END_VAR
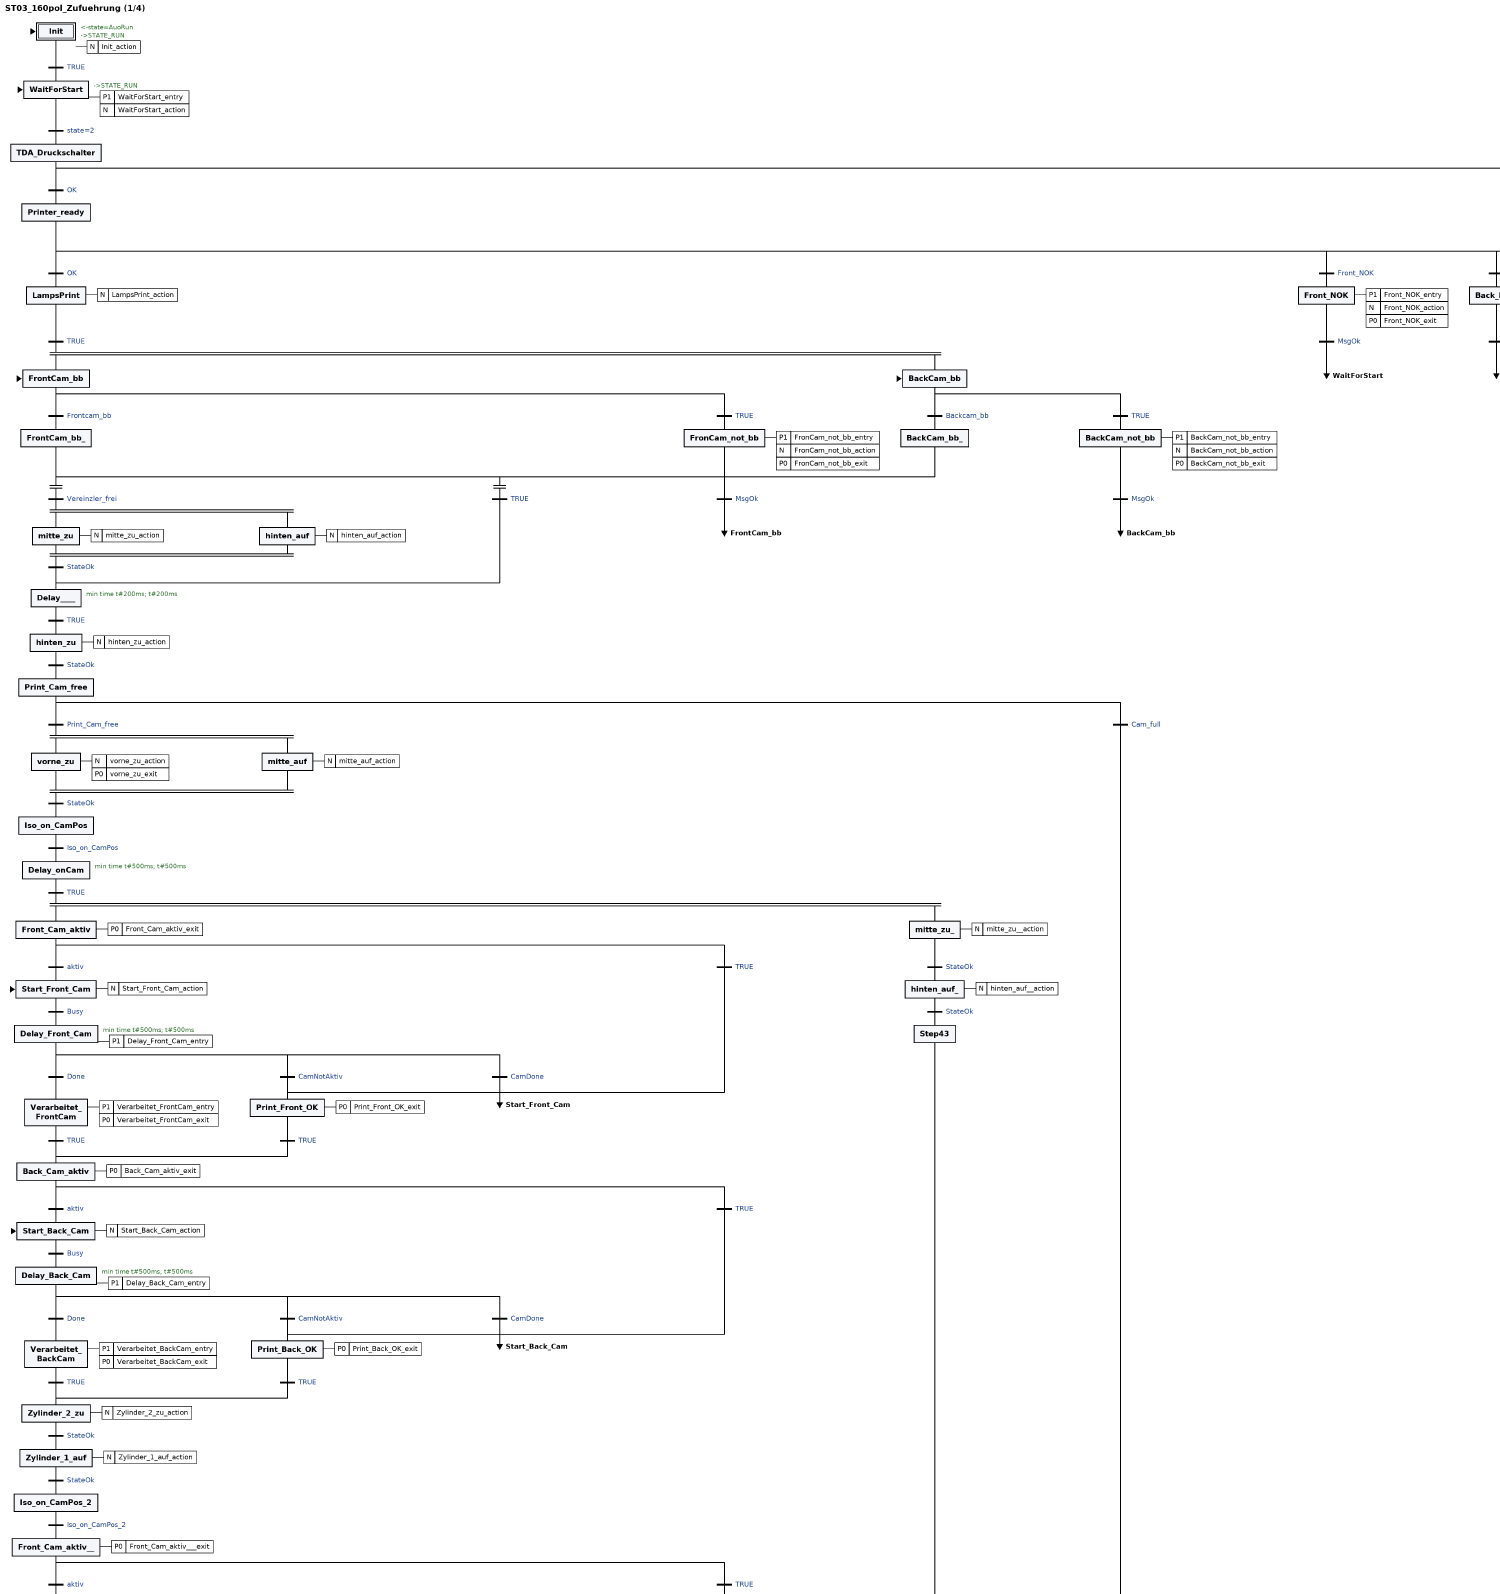
[picture p37: ST03_160pol_Zufuehrung (SFC)]
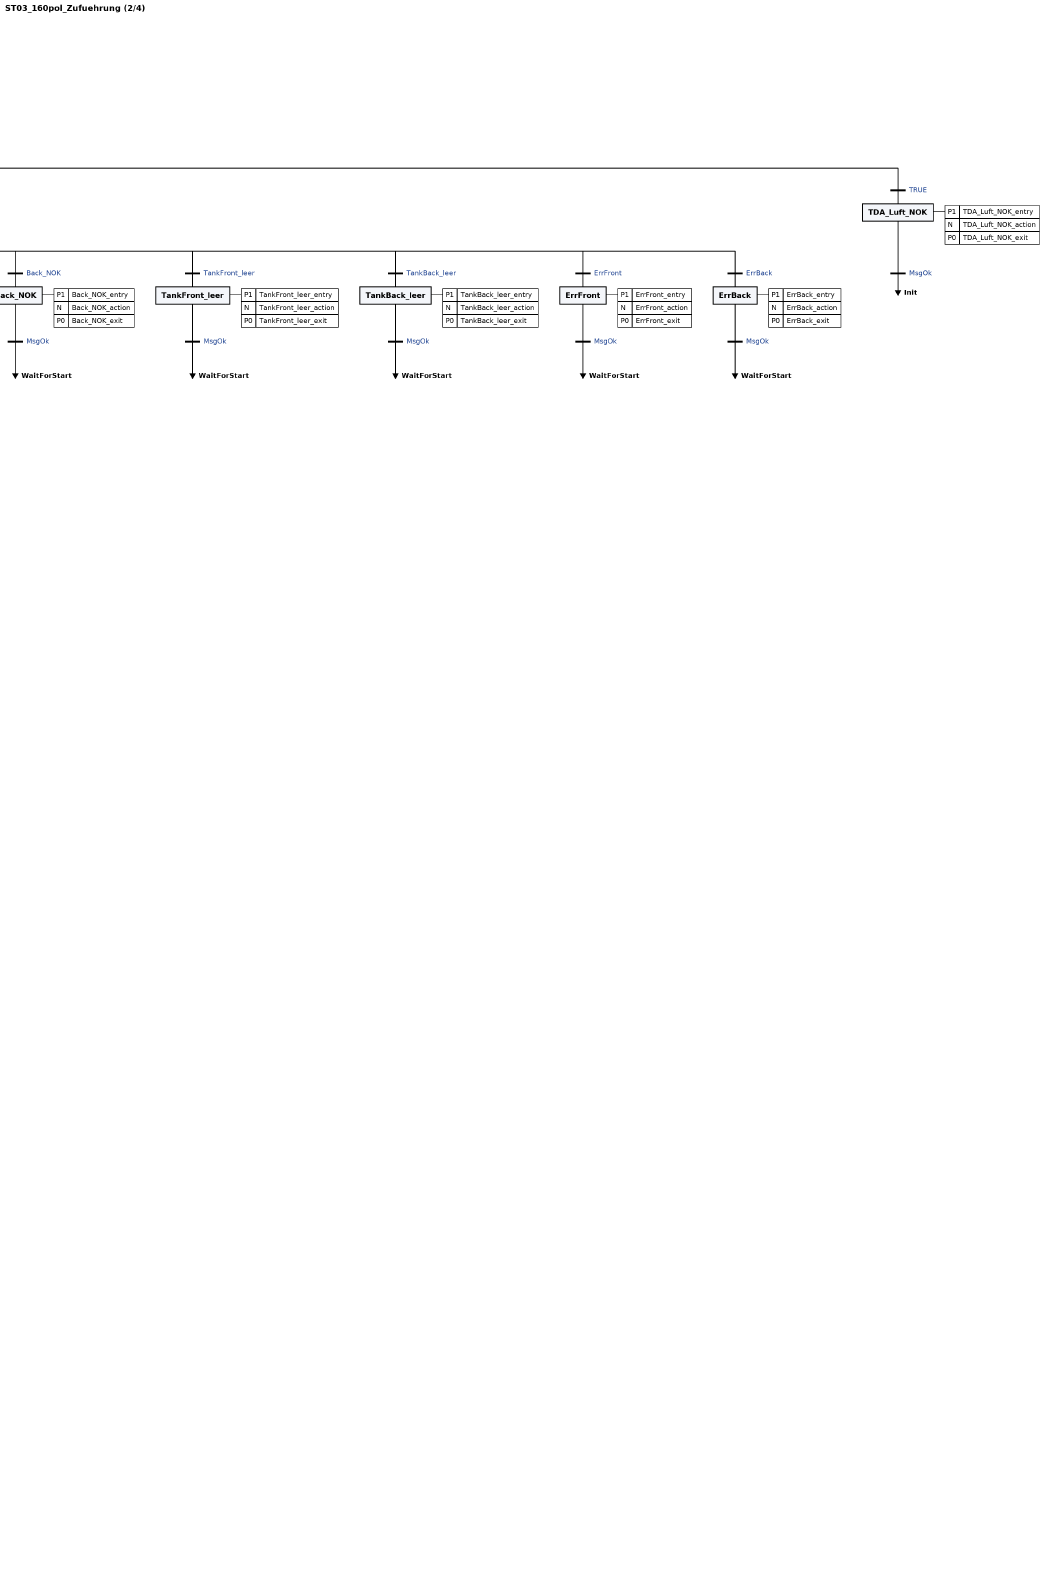
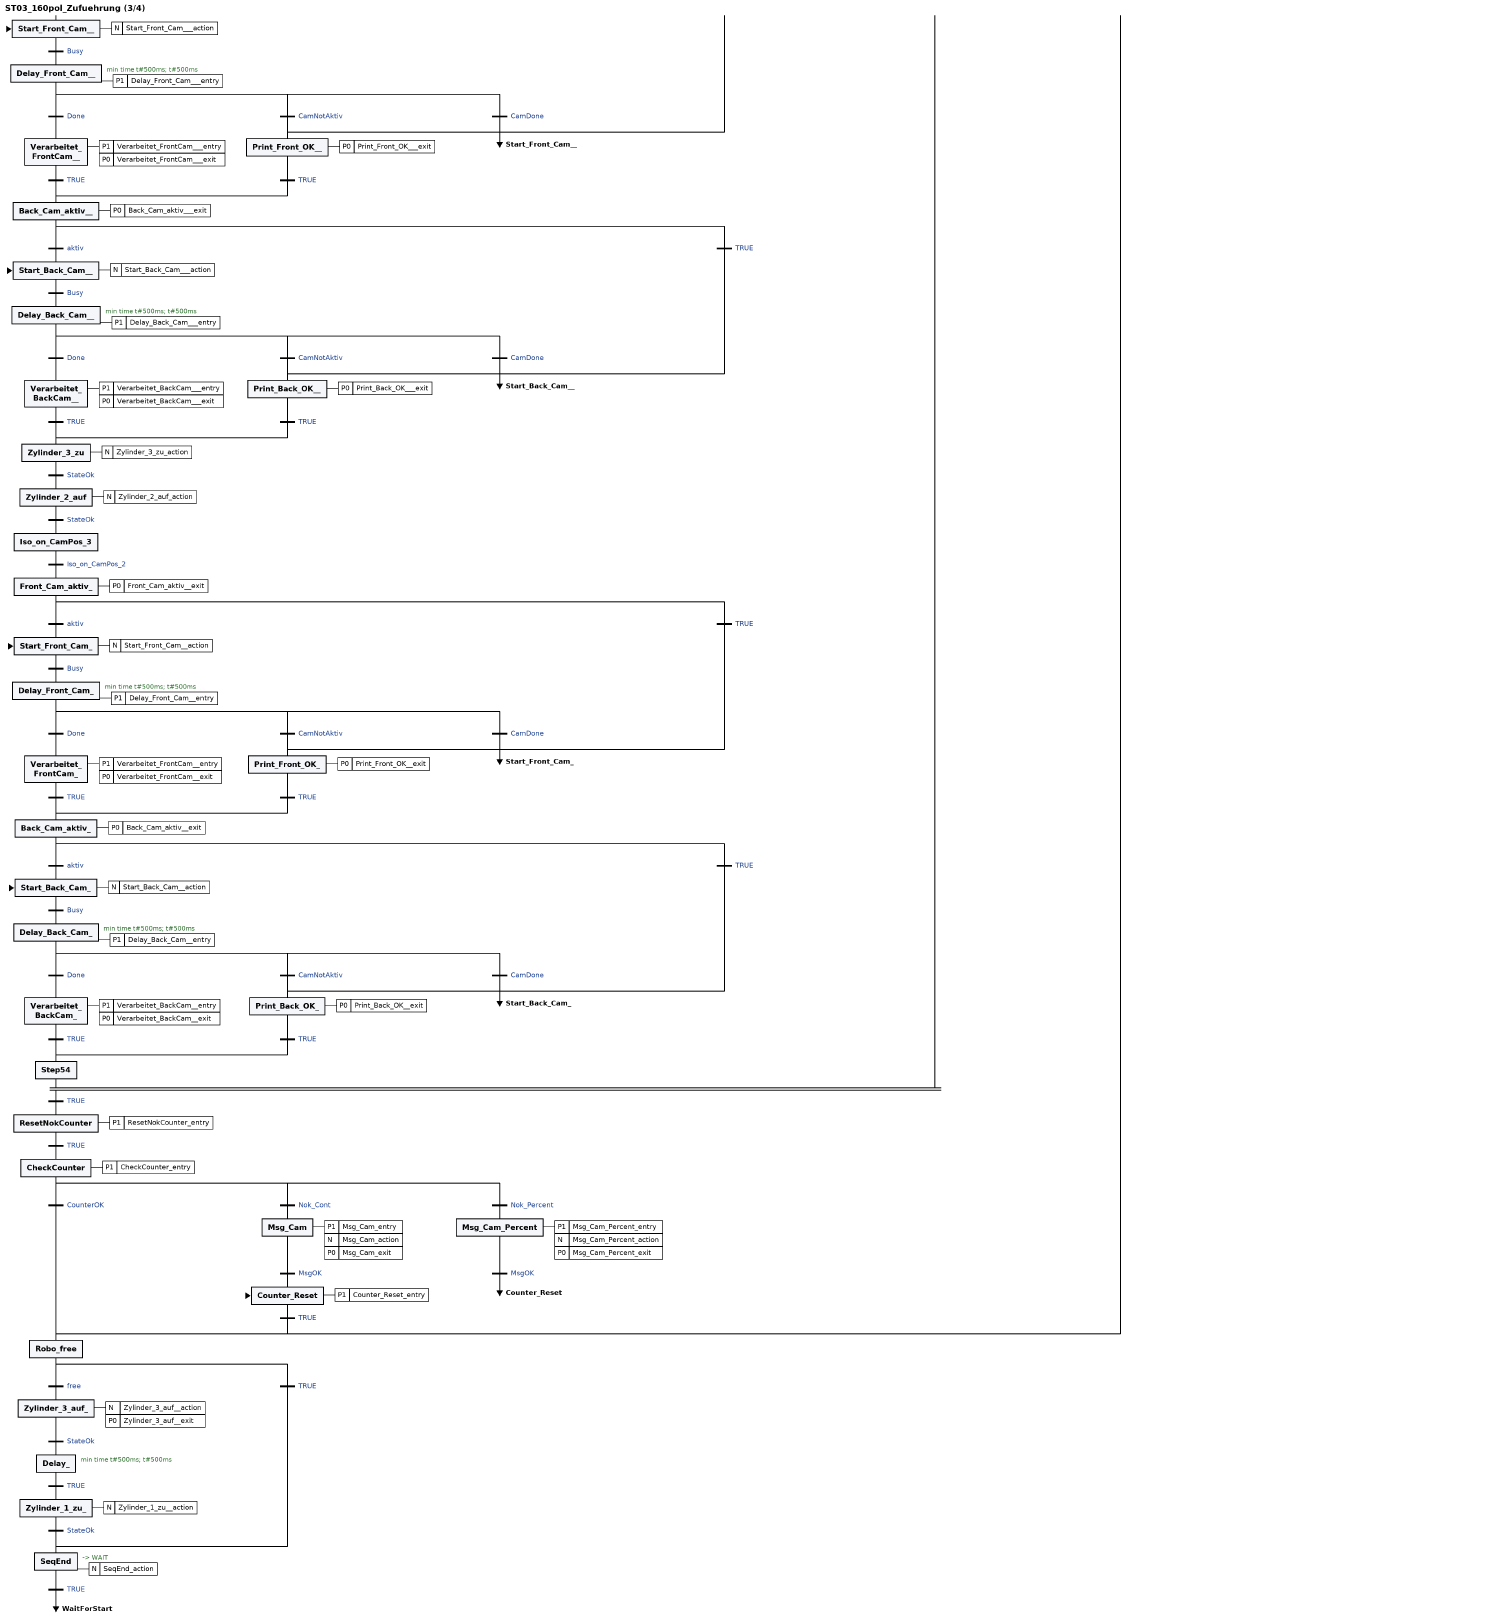
INITIAL_STEP Init: (* <-state=AuoRun / ->STATE_RUN *)
	Init_action(N);
END_STEP
TRANSITION FROM Init TO WaitForStart := TRUE;
END_TRANSITION
STEP WaitForStart: (* ->STATE_RUN *)
	WaitForStart_entry(P1);
	WaitForStart_action(N);
END_STEP
TRANSITION FROM WaitForStart TO TDA_Druckschalter := state=2;
END_TRANSITION
STEP TDA_Druckschalter:
END_STEP
TRANSITION FROM TDA_Druckschalter TO Printer_ready := OK;
END_TRANSITION
TRANSITION FROM TDA_Druckschalter TO TDA_Luft_NOK := TRUE;
END_TRANSITION
STEP TDA_Luft_NOK:
	TDA_Luft_NOK_entry(P1);
	TDA_Luft_NOK_action(N);
	TDA_Luft_NOK_exit(P0);
END_STEP
TRANSITION FROM TDA_Luft_NOK TO Init := MsgOk;
END_TRANSITION
STEP Printer_ready:
END_STEP
TRANSITION FROM Printer_ready TO LampsPrint := OK;
END_TRANSITION
TRANSITION FROM Printer_ready TO Front_NOK := Front_NOK;
END_TRANSITION
TRANSITION FROM Printer_ready TO Back_NOK := Back_NOK;
END_TRANSITION
TRANSITION FROM Printer_ready TO TankFront_leer := TankFront_leer;
END_TRANSITION
TRANSITION FROM Printer_ready TO TankBack_leer := TankBack_leer;
END_TRANSITION
TRANSITION FROM Printer_ready TO ErrFront := ErrFront;
END_TRANSITION
TRANSITION FROM Printer_ready TO ErrBack := ErrBack;
END_TRANSITION
STEP LampsPrint:
	LampsPrint_action(N);
END_STEP
TRANSITION FROM LampsPrint TO (FrontCam_bb, BackCam_bb) := TRUE;
END_TRANSITION
STEP Front_NOK:
	Front_NOK_entry(P1);
	Front_NOK_action(N);
	Front_NOK_exit(P0);
END_STEP
TRANSITION FROM Front_NOK TO WaitForStart := MsgOk;
END_TRANSITION
STEP Back_NOK:
	Back_NOK_entry(P1);
	Back_NOK_action(N);
	Back_NOK_exit(P0);
END_STEP
TRANSITION FROM Back_NOK TO WaitForStart := MsgOk;
END_TRANSITION
STEP TankFront_leer:
	TankFront_leer_entry(P1);
	TankFront_leer_action(N);
	TankFront_leer_exit(P0);
END_STEP
TRANSITION FROM TankFront_leer TO WaitForStart := MsgOk;
END_TRANSITION
STEP TankBack_leer:
	TankBack_leer_entry(P1);
	TankBack_leer_action(N);
	TankBack_leer_exit(P0);
END_STEP
TRANSITION FROM TankBack_leer TO WaitForStart := MsgOk;
END_TRANSITION
STEP ErrFront:
	ErrFront_entry(P1);
	ErrFront_action(N);
	ErrFront_exit(P0);
END_STEP
TRANSITION FROM ErrFront TO WaitForStart := MsgOk;
END_TRANSITION
STEP ErrBack:
	ErrBack_entry(P1);
	ErrBack_action(N);
	ErrBack_exit(P0);
END_STEP
TRANSITION FROM ErrBack TO WaitForStart := MsgOk;
END_TRANSITION
STEP FrontCam_bb:
END_STEP
TRANSITION FROM FrontCam_bb TO FrontCam_bb_ := Frontcam_bb;
END_TRANSITION
TRANSITION FROM FrontCam_bb TO FronCam_not_bb := TRUE;
END_TRANSITION
STEP FronCam_not_bb:
	FronCam_not_bb_entry(P1);
	FronCam_not_bb_action(N);
	FronCam_not_bb_exit(P0);
END_STEP
TRANSITION FROM FronCam_not_bb TO FrontCam_bb := MsgOk;
END_TRANSITION
STEP FrontCam_bb_:
END_STEP
STEP BackCam_bb:
END_STEP
TRANSITION FROM BackCam_bb TO BackCam_bb_ := Backcam_bb;
END_TRANSITION
TRANSITION FROM BackCam_bb TO BackCam_not_bb := TRUE;
END_TRANSITION
STEP BackCam_not_bb:
	BackCam_not_bb_entry(P1);
	BackCam_not_bb_action(N);
	BackCam_not_bb_exit(P0);
END_STEP
TRANSITION FROM BackCam_not_bb TO BackCam_bb := MsgOk;
END_TRANSITION
STEP BackCam_bb_:
END_STEP
TRANSITION FROM (FrontCam_bb_, BackCam_bb_) TO (mitte_zu, hinten_auf) := Vereinzler_frei;
END_TRANSITION
TRANSITION FROM (FrontCam_bb_, BackCam_bb_) TO Delay____ := TRUE;
END_TRANSITION
STEP mitte_zu:
	mitte_zu_action(N);
END_STEP
STEP hinten_auf:
	hinten_auf_action(N);
END_STEP
TRANSITION FROM (mitte_zu, hinten_auf) TO Delay____ := StateOk;
END_TRANSITION
STEP Delay____: (* min time t#200ms; t#200ms *)
END_STEP
TRANSITION FROM Delay____ TO hinten_zu := TRUE;
END_TRANSITION
STEP hinten_zu:
	hinten_zu_action(N);
END_STEP
TRANSITION FROM hinten_zu TO Print_Cam_free := StateOk;
END_TRANSITION
STEP Print_Cam_free:
END_STEP
TRANSITION FROM Print_Cam_free TO (vorne_zu, mitte_auf) := Print_Cam_free;
END_TRANSITION
TRANSITION FROM Print_Cam_free TO Robo_free := Cam_full;
END_TRANSITION
STEP vorne_zu:
	vorne_zu_action(N);
	vorne_zu_exit(P0);
END_STEP
STEP mitte_auf:
	mitte_auf_action(N);
END_STEP
TRANSITION FROM (vorne_zu, mitte_auf) TO Iso_on_CamPos := StateOk;
END_TRANSITION
STEP Iso_on_CamPos:
END_STEP
TRANSITION FROM Iso_on_CamPos TO Delay_onCam := Iso_on_CamPos;
END_TRANSITION
STEP Delay_onCam: (* min time t#500ms; t#500ms *)
END_STEP
TRANSITION FROM Delay_onCam TO (Front_Cam_aktiv, mitte_zu_) := TRUE;
END_TRANSITION
STEP Front_Cam_aktiv:
	Front_Cam_aktiv_exit(P0);
END_STEP
TRANSITION FROM Front_Cam_aktiv TO Start_Front_Cam := aktiv;
END_TRANSITION
TRANSITION FROM Front_Cam_aktiv TO Print_Front_OK := TRUE;
END_TRANSITION
STEP Start_Front_Cam:
	Start_Front_Cam_action(N);
END_STEP
TRANSITION FROM Start_Front_Cam TO Delay_Front_Cam := Busy;
END_TRANSITION
STEP Delay_Front_Cam: (* min time t#500ms; t#500ms *)
	Delay_Front_Cam_entry(P1);
END_STEP
TRANSITION FROM Delay_Front_Cam TO Verarbeitet_FrontCam := Done;
END_TRANSITION
TRANSITION FROM Delay_Front_Cam TO Print_Front_OK := CamNotAktiv;
END_TRANSITION
TRANSITION FROM Delay_Front_Cam TO Start_Front_Cam := CamDone;
END_TRANSITION
STEP Verarbeitet_FrontCam:
	Verarbeitet_FrontCam_entry(P1);
	Verarbeitet_FrontCam_exit(P0);
END_STEP
TRANSITION FROM Verarbeitet_FrontCam TO Back_Cam_aktiv := TRUE;
END_TRANSITION
STEP Print_Front_OK:
	Print_Front_OK_exit(P0);
END_STEP
TRANSITION FROM Print_Front_OK TO Back_Cam_aktiv := TRUE;
END_TRANSITION
STEP Back_Cam_aktiv:
	Back_Cam_aktiv_exit(P0);
END_STEP
TRANSITION FROM Back_Cam_aktiv TO Start_Back_Cam := aktiv;
END_TRANSITION
TRANSITION FROM Back_Cam_aktiv TO Print_Back_OK := TRUE;
END_TRANSITION
STEP Start_Back_Cam:
	Start_Back_Cam_action(N);
END_STEP
TRANSITION FROM Start_Back_Cam TO Delay_Back_Cam := Busy;
END_TRANSITION
STEP Delay_Back_Cam: (* min time t#500ms; t#500ms *)
	Delay_Back_Cam_entry(P1);
END_STEP
TRANSITION FROM Delay_Back_Cam TO Verarbeitet_BackCam := Done;
END_TRANSITION
TRANSITION FROM Delay_Back_Cam TO Print_Back_OK := CamNotAktiv;
END_TRANSITION
TRANSITION FROM Delay_Back_Cam TO Start_Back_Cam := CamDone;
END_TRANSITION
STEP Verarbeitet_BackCam:
	Verarbeitet_BackCam_entry(P1);
	Verarbeitet_BackCam_exit(P0);
END_STEP
TRANSITION FROM Verarbeitet_BackCam TO Zylinder_2_zu := TRUE;
END_TRANSITION
STEP Print_Back_OK:
	Print_Back_OK_exit(P0);
END_STEP
TRANSITION FROM Print_Back_OK TO Zylinder_2_zu := TRUE;
END_TRANSITION
STEP Zylinder_2_zu:
	Zylinder_2_zu_action(N);
END_STEP
TRANSITION FROM Zylinder_2_zu TO Zylinder_1_auf := StateOk;
END_TRANSITION
STEP Zylinder_1_auf:
	Zylinder_1_auf_action(N);
END_STEP
TRANSITION FROM Zylinder_1_auf TO Iso_on_CamPos_2 := StateOk;
END_TRANSITION
STEP Iso_on_CamPos_2:
END_STEP
TRANSITION FROM Iso_on_CamPos_2 TO Front_Cam_aktiv__ := Iso_on_CamPos_2;
END_TRANSITION
STEP Front_Cam_aktiv__:
	Front_Cam_aktiv___exit(P0);
END_STEP
TRANSITION FROM Front_Cam_aktiv__ TO Start_Front_Cam__ := aktiv;
END_TRANSITION
TRANSITION FROM Front_Cam_aktiv__ TO Print_Front_OK__ := TRUE;
END_TRANSITION
STEP Start_Front_Cam__:
	Start_Front_Cam___action(N);
END_STEP
TRANSITION FROM Start_Front_Cam__ TO Delay_Front_Cam__ := Busy;
END_TRANSITION
STEP Delay_Front_Cam__: (* min time t#500ms; t#500ms *)
	Delay_Front_Cam___entry(P1);
END_STEP
TRANSITION FROM Delay_Front_Cam__ TO Verarbeitet_FrontCam__ := Done;
END_TRANSITION
TRANSITION FROM Delay_Front_Cam__ TO Print_Front_OK__ := CamNotAktiv;
END_TRANSITION
TRANSITION FROM Delay_Front_Cam__ TO Start_Front_Cam__ := CamDone;
END_TRANSITION
STEP Verarbeitet_FrontCam__:
	Verarbeitet_FrontCam___entry(P1);
	Verarbeitet_FrontCam___exit(P0);
END_STEP
TRANSITION FROM Verarbeitet_FrontCam__ TO Back_Cam_aktiv__ := TRUE;
END_TRANSITION
STEP Print_Front_OK__:
	Print_Front_OK___exit(P0);
END_STEP
TRANSITION FROM Print_Front_OK__ TO Back_Cam_aktiv__ := TRUE;
END_TRANSITION
STEP Back_Cam_aktiv__:
	Back_Cam_aktiv___exit(P0);
END_STEP
TRANSITION FROM Back_Cam_aktiv__ TO Start_Back_Cam__ := aktiv;
END_TRANSITION
TRANSITION FROM Back_Cam_aktiv__ TO Print_Back_OK__ := TRUE;
END_TRANSITION
STEP Start_Back_Cam__:
	Start_Back_Cam___action(N);
END_STEP
TRANSITION FROM Start_Back_Cam__ TO Delay_Back_Cam__ := Busy;
END_TRANSITION
STEP Delay_Back_Cam__: (* min time t#500ms; t#500ms *)
	Delay_Back_Cam___entry(P1);
END_STEP
TRANSITION FROM Delay_Back_Cam__ TO Verarbeitet_BackCam__ := Done;
END_TRANSITION
TRANSITION FROM Delay_Back_Cam__ TO Print_Back_OK__ := CamNotAktiv;
END_TRANSITION
TRANSITION FROM Delay_Back_Cam__ TO Start_Back_Cam__ := CamDone;
END_TRANSITION
STEP Verarbeitet_BackCam__:
	Verarbeitet_BackCam___entry(P1);
	Verarbeitet_BackCam___exit(P0);
END_STEP
TRANSITION FROM Verarbeitet_BackCam__ TO Zylinder_3_zu := TRUE;
END_TRANSITION
STEP Print_Back_OK__:
	Print_Back_OK___exit(P0);
END_STEP
TRANSITION FROM Print_Back_OK__ TO Zylinder_3_zu := TRUE;
END_TRANSITION
STEP Zylinder_3_zu:
	Zylinder_3_zu_action(N);
END_STEP
TRANSITION FROM Zylinder_3_zu TO Zylinder_2_auf := StateOk;
END_TRANSITION
STEP Zylinder_2_auf:
	Zylinder_2_auf_action(N);
END_STEP
TRANSITION FROM Zylinder_2_auf TO Iso_on_CamPos_3 := StateOk;
END_TRANSITION
STEP Iso_on_CamPos_3:
END_STEP
TRANSITION FROM Iso_on_CamPos_3 TO Front_Cam_aktiv_ := Iso_on_CamPos_2;
END_TRANSITION
STEP Front_Cam_aktiv_:
	Front_Cam_aktiv__exit(P0);
END_STEP
TRANSITION FROM Front_Cam_aktiv_ TO Start_Front_Cam_ := aktiv;
END_TRANSITION
TRANSITION FROM Front_Cam_aktiv_ TO Print_Front_OK_ := TRUE;
END_TRANSITION
STEP Start_Front_Cam_:
	Start_Front_Cam__action(N);
END_STEP
TRANSITION FROM Start_Front_Cam_ TO Delay_Front_Cam_ := Busy;
END_TRANSITION
STEP Delay_Front_Cam_: (* min time t#500ms; t#500ms *)
	Delay_Front_Cam__entry(P1);
END_STEP
TRANSITION FROM Delay_Front_Cam_ TO Verarbeitet_FrontCam_ := Done;
END_TRANSITION
TRANSITION FROM Delay_Front_Cam_ TO Print_Front_OK_ := CamNotAktiv;
END_TRANSITION
TRANSITION FROM Delay_Front_Cam_ TO Start_Front_Cam_ := CamDone;
END_TRANSITION
STEP Verarbeitet_FrontCam_:
	Verarbeitet_FrontCam__entry(P1);
	Verarbeitet_FrontCam__exit(P0);
END_STEP
TRANSITION FROM Verarbeitet_FrontCam_ TO Back_Cam_aktiv_ := TRUE;
END_TRANSITION
STEP Print_Front_OK_:
	Print_Front_OK__exit(P0);
END_STEP
TRANSITION FROM Print_Front_OK_ TO Back_Cam_aktiv_ := TRUE;
END_TRANSITION
STEP Back_Cam_aktiv_:
	Back_Cam_aktiv__exit(P0);
END_STEP
TRANSITION FROM Back_Cam_aktiv_ TO Start_Back_Cam_ := aktiv;
END_TRANSITION
TRANSITION FROM Back_Cam_aktiv_ TO Print_Back_OK_ := TRUE;
END_TRANSITION
STEP Start_Back_Cam_:
	Start_Back_Cam__action(N);
END_STEP
TRANSITION FROM Start_Back_Cam_ TO Delay_Back_Cam_ := Busy;
END_TRANSITION
STEP Delay_Back_Cam_: (* min time t#500ms; t#500ms *)
	Delay_Back_Cam__entry(P1);
END_STEP
TRANSITION FROM Delay_Back_Cam_ TO Verarbeitet_BackCam_ := Done;
END_TRANSITION
TRANSITION FROM Delay_Back_Cam_ TO Print_Back_OK_ := CamNotAktiv;
END_TRANSITION
TRANSITION FROM Delay_Back_Cam_ TO Start_Back_Cam_ := CamDone;
END_TRANSITION
STEP Verarbeitet_BackCam_:
	Verarbeitet_BackCam__entry(P1);
	Verarbeitet_BackCam__exit(P0);
END_STEP
TRANSITION FROM Verarbeitet_BackCam_ TO Step54 := TRUE;
END_TRANSITION
STEP Print_Back_OK_:
	Print_Back_OK__exit(P0);
END_STEP
TRANSITION FROM Print_Back_OK_ TO Step54 := TRUE;
END_TRANSITION
STEP Step54:
END_STEP
STEP mitte_zu_:
	mitte_zu__action(N);
END_STEP
TRANSITION FROM mitte_zu_ TO hinten_auf_ := StateOk;
END_TRANSITION
STEP hinten_auf_:
	hinten_auf__action(N);
END_STEP
TRANSITION FROM hinten_auf_ TO Step43 := StateOk;
END_TRANSITION
STEP Step43:
END_STEP
TRANSITION FROM (Step54, Step43) TO ResetNokCounter := TRUE;
END_TRANSITION
STEP ResetNokCounter:
	ResetNokCounter_entry(P1);
END_STEP
TRANSITION FROM ResetNokCounter TO CheckCounter := TRUE;
END_TRANSITION
STEP CheckCounter:
	CheckCounter_entry(P1);
END_STEP
TRANSITION FROM CheckCounter TO Robo_free := CounterOK;
END_TRANSITION
TRANSITION FROM CheckCounter TO Msg_Cam := Nok_Cont;
END_TRANSITION
TRANSITION FROM CheckCounter TO Msg_Cam_Percent := Nok_Percent;
END_TRANSITION
STEP Msg_Cam:
	Msg_Cam_entry(P1);
	Msg_Cam_action(N);
	Msg_Cam_exit(P0);
END_STEP
TRANSITION FROM Msg_Cam TO Counter_Reset := MsgOK;
END_TRANSITION
STEP Counter_Reset:
	Counter_Reset_entry(P1);
END_STEP
TRANSITION FROM Counter_Reset TO Robo_free := TRUE;
END_TRANSITION
STEP Msg_Cam_Percent:
	Msg_Cam_Percent_entry(P1);
	Msg_Cam_Percent_action(N);
	Msg_Cam_Percent_exit(P0);
END_STEP
TRANSITION FROM Msg_Cam_Percent TO Counter_Reset := MsgOK;
END_TRANSITION
STEP Robo_free:
END_STEP
TRANSITION FROM Robo_free TO Zylinder_3_auf_ := free;
END_TRANSITION
TRANSITION FROM Robo_free TO SeqEnd := TRUE;
END_TRANSITION
STEP Zylinder_3_auf_:
	Zylinder_3_auf__action(N);
	Zylinder_3_auf__exit(P0);
END_STEP
TRANSITION FROM Zylinder_3_auf_ TO Delay_ := StateOk;
END_TRANSITION
STEP Delay_: (* min time t#500ms; t#500ms *)
END_STEP
TRANSITION FROM Delay_ TO Zylinder_1_zu_ := TRUE;
END_TRANSITION
STEP Zylinder_1_zu_:
	Zylinder_1_zu__action(N);
END_STEP
TRANSITION FROM Zylinder_1_zu_ TO SeqEnd := StateOk;
END_TRANSITION
STEP SeqEnd: (* -> WAIT *)
	SeqEnd_action(N);
END_STEP
TRANSITION FROM SeqEnd TO WaitForStart := TRUE;
END_TRANSITION

ACTION Init_action:
Start:=FALSE;
State:=STATE_WAIT;
MsgOK:=FALSE;
MsgCancel:=FALSE;
SFCRun:=FALSE;
Result160pol:=RESULT_NON;
NokCounter:=0;

ST03_8_80_A1.b_start := FALSE;
ST03_8_85_A1.b_start := FALSE;

ST03_8_90_A1.st_ctrl_in.b_start := FALSE;
ST03_8_95_A1.st_ctrl_in.b_start := FALSE;
END_ACTION

ACTION WaitForStart_entry:
;
END_ACTION

ACTION WaitForStart_action:
IF 	Start   THEN
	State:=STATE_RUN;
	SFCTimeStart:=TIME();
	Start:=FALSE;
ELSE
	State:=STATE_WAIT;
	MsgOK:=FALSE;
	MsgCancel:=FALSE;
	SFCRun:=FALSE;
END_IF
END_ACTION

ACTION TDA_Luft_NOK_entry:
MessageHandler.ClearMessageLines(sVisu:=Visu.Message);
END_ACTION

ACTION TDA_Luft_NOK_action:
MessageHandler.Msg.ID:='PM103';
MessageHandler.Msg.Name:='Tintenstrahldrucker Druckschalter';
MessageHandler.Msg.Text:='ST02 Druckschalter Wartungseinheit Hauptluft min.6 bar';
MessageHandler.Msg.Color:=Color.red;
MessageHandler.Msg.Station:=1;


MessageHandler(
	Prio:=2, 							(*1=highest, .. , 4=lowest*)
	Btn1Addr:=ADR(MsgOk),			(*Address of Button1 , if Zero then Button is unvisible*)
	Btn2Addr:=,						(*Address of Button2 , if Zero then Button is unvisible*)
	sVisu:=Visu.Message);
END_ACTION

ACTION TDA_Luft_NOK_exit:
MsgOk:=FALSE;
MsgCancel:=FALSE;
END_ACTION

ACTION LampsPrint_action:
(*Signalsäule Tintenstrahldrucker schalten, nur bei SGM-3621*)

(*Signalsäuele Bedruckung RD Sammelstörung*)
ST03_H7.SetSignalHigh:= FALSE;
ST03_H7.SetSignalLow:= TRUE;
(*Signalsäule Bedruckung GR Bedruckung IO*)
ST03_H6.SetSignalHigh:= TRUE;
ST03_H6.SetSignalLow:= FALSE;
END_ACTION

ACTION Front_NOK_entry:
MessageHandler.ClearMessageLines(sVisu:=Visu.Message);
END_ACTION

ACTION Front_NOK_action:
MessageHandler.Msg.ID:='PM104';
MessageHandler.Msg.Name:=ST03_70U3_1.sInit.Description;
MessageHandler.Msg.Text:='Drucker Front nicht betriebsbereit';
MessageHandler.Msg.Color:=Color.red;
MessageHandler.Msg.Station:=1;


MessageHandler(
	Prio:=2, 							(*1=highest, .. , 4=lowest*)
	Btn1Addr:=ADR(MsgOk),			(*Address of Button1 , if Zero then Button is unvisible*)
	Btn2Addr:=,						(*Address of Button2 , if Zero then Button is unvisible*)
	sVisu:=Visu.Message);
END_ACTION

ACTION Front_NOK_exit:
MsgOk:=FALSE;
MsgCancel:=FALSE;
END_ACTION

ACTION Back_NOK_entry:
MessageHandler.ClearMessageLines(sVisu:=Visu.Message);
END_ACTION

ACTION Back_NOK_action:
MessageHandler.Msg.ID:='PM105';
MessageHandler.Msg.Name:=ST03_71U3_1.sInit.Description;
MessageHandler.Msg.Text:='Drucker Rückseite nicht betriebsbereit';
MessageHandler.Msg.Color:=Color.red;
MessageHandler.Msg.Station:=1;


MessageHandler(
	Prio:=2, 							(*1=highest, .. , 4=lowest*)
	Btn1Addr:=ADR(MsgOk),			(*Address of Button1 , if Zero then Button is unvisible*)
	Btn2Addr:=,						(*Address of Button2 , if Zero then Button is unvisible*)
	sVisu:=Visu.Message);
END_ACTION

ACTION Back_NOK_exit:
MsgOk:=FALSE;
MsgCancel:=FALSE;
END_ACTION

ACTION TankFront_leer_entry:
MessageHandler.ClearMessageLines(sVisu:=Visu.Message);
END_ACTION

ACTION TankFront_leer_action:
MessageHandler.Msg.ID:='PM106';
MessageHandler.Msg.Name:=ST03_70U3_2.sInit.Description;
MessageHandler.Msg.Text:='Tank Drucker Frontseite leer';
MessageHandler.Msg.Color:=Color.red;
MessageHandler.Msg.Station:=1;


MessageHandler(
	Prio:=2, 							(*1=highest, .. , 4=lowest*)
	Btn1Addr:=ADR(MsgOk),			(*Address of Button1 , if Zero then Button is unvisible*)
	Btn2Addr:=,						(*Address of Button2 , if Zero then Button is unvisible*)
	sVisu:=Visu.Message);
END_ACTION

ACTION TankFront_leer_exit:
MsgOk:=FALSE;
MsgCancel:=FALSE;
END_ACTION

ACTION TankBack_leer_entry:
MessageHandler.ClearMessageLines(sVisu:=Visu.Message);
END_ACTION

ACTION TankBack_leer_action:
MessageHandler.Msg.ID:='PM107';
MessageHandler.Msg.Name:=ST03_71U3_2.sInit.Description;
MessageHandler.Msg.Text:='Tank Drucker Rückseite leer';
MessageHandler.Msg.Color:=Color.red;
MessageHandler.Msg.Station:=1;


MessageHandler(
	Prio:=2, 							(*1=highest, .. , 4=lowest*)
	Btn1Addr:=ADR(MsgOk),			(*Address of Button1 , if Zero then Button is unvisible*)
	Btn2Addr:=,						(*Address of Button2 , if Zero then Button is unvisible*)
	sVisu:=Visu.Message);
END_ACTION

ACTION TankBack_leer_exit:
MsgOk:=FALSE;
MsgCancel:=FALSE;
END_ACTION

ACTION ErrFront_entry:
MessageHandler.ClearMessageLines(sVisu:=Visu.Message);
(*Signalsäuele Bedruckung RD Sammelstörung*)
ST03_H7.SetSignalHigh:= TRUE;
ST03_H7.SetSignalLow:= FALSE;
(*Signalsäule Bedruckung GR Bedruckung IO*)
ST03_H6.SetSignalHigh:= FALSE;
ST03_H6.SetSignalLow:= TRUE;
END_ACTION

ACTION ErrFront_action:
MessageHandler.Msg.ID:='PM108';
MessageHandler.Msg.Name:=ST03_70U3_3.sInit.Description;
MessageHandler.Msg.Text:='Störung Drucker Frontseite ';
MessageHandler.Msg.Color:=Color.red;
MessageHandler.Msg.Station:=1;


MessageHandler(
	Prio:=2, 							(*1=highest, .. , 4=lowest*)
	Btn1Addr:=ADR(MsgOk),			(*Address of Button1 , if Zero then Button is unvisible*)
	Btn2Addr:=,						(*Address of Button2 , if Zero then Button is unvisible*)
	sVisu:=Visu.Message);
END_ACTION

ACTION ErrFront_exit:
MsgOk:=FALSE;
MsgCancel:=FALSE;
(*Signalsäuele Bedruckung RD Sammelstörung*)
ST03_H7.SetSignalHigh:= FALSE;
ST03_H7.SetSignalLow:= TRUE;
(*Signalsäule Bedruckung GR Bedruckung IO*)
ST03_H6.SetSignalHigh:= TRUE;
ST03_H6.SetSignalLow:= FALSE;
END_ACTION

ACTION ErrBack_entry:
MessageHandler.ClearMessageLines(sVisu:=Visu.Message);
(*Signalsäuele Bedruckung RD Sammelstörung*)
ST03_H7.SetSignalHigh:= TRUE;
ST03_H7.SetSignalLow:= FALSE;
(*Signalsäule Bedruckung GR Bedruckung IO*)
ST03_H6.SetSignalHigh:= FALSE;
ST03_H6.SetSignalLow:= TRUE;
END_ACTION

ACTION ErrBack_action:
MessageHandler.Msg.ID:='PM109';
MessageHandler.Msg.Name:=ST03_71U3_3.sInit.Description;
MessageHandler.Msg.Text:='Störung Drucker Rückseite';
MessageHandler.Msg.Color:=Color.red;
MessageHandler.Msg.Station:=1;


MessageHandler(
	Prio:=2, 							(*1=highest, .. , 4=lowest*)
	Btn1Addr:=ADR(MsgOk),			(*Address of Button1 , if Zero then Button is unvisible*)
	Btn2Addr:=,						(*Address of Button2 , if Zero then Button is unvisible*)
	sVisu:=Visu.Message);
END_ACTION

ACTION ErrBack_exit:
MsgOk:=FALSE;
MsgCancel:=FALSE;
(*Signalsäuele Bedruckung RD Sammelstörung*)
ST03_H7.SetSignalHigh:= FALSE;
ST03_H7.SetSignalLow:= TRUE;
(*Signalsäule Bedruckung GR Bedruckung IO*)
ST03_H6.SetSignalHigh:= TRUE;
ST03_H6.SetSignalLow:= FALSE;
END_ACTION

ACTION FronCam_not_bb_entry:
MessageHandler.ClearMessageLines(sVisu:=Visu.Message);
END_ACTION

ACTION FronCam_not_bb_action:
MessageHandler.Msg.ID:='PM110';
MessageHandler.Msg.Name:='Check Camera';
MessageHandler.Msg.Text:='Kamera Frontseite ist nicht betriebsbereit';
MessageHandler.Msg.Color:=Color.red;
MessageHandler.Msg.Station:=1;


MessageHandler(
	Prio:=2, 							(*1=highest, .. , 4=lowest*)
	Btn1Addr:=ADR(MsgOk),			(*Address of Button1 , if Zero then Button is unvisible*)
	Btn2Addr:=,						(*Address of Button2 , if Zero then Button is unvisible*)
	sVisu:=Visu.Message);
END_ACTION

ACTION FronCam_not_bb_exit:
MsgOk:=FALSE;
MsgCancel:=FALSE;
END_ACTION

ACTION BackCam_not_bb_entry:
MessageHandler.ClearMessageLines(sVisu:=Visu.Message);
END_ACTION

ACTION BackCam_not_bb_action:
MessageHandler.Msg.ID:='PM111';
MessageHandler.Msg.Name:='Check Camera';
MessageHandler.Msg.Text:='Kamera Rückseite ist nicht betriebsbereit';
MessageHandler.Msg.Color:=Color.red;
MessageHandler.Msg.Station:=1;


MessageHandler(
	Prio:=2, 							(*1=highest, .. , 4=lowest*)
	Btn1Addr:=ADR(MsgOk),			(*Address of Button1 , if Zero then Button is unvisible*)
	Btn2Addr:=,						(*Address of Button2 , if Zero then Button is unvisible*)
	sVisu:=Visu.Message);
END_ACTION

ACTION BackCam_not_bb_exit:
MsgOk:=FALSE;
MsgCancel:=FALSE;
END_ACTION

ACTION mitte_zu_action:
ST03_422_Y64_6.MoveInit:=TRUE;	(* Förderband  Stopper Vereinzler AST/GST *)
END_ACTION

ACTION hinten_auf_action:
ST03_422_Y64_5.MoveInit:=TRUE;
END_ACTION

ACTION hinten_zu_action:
ST03_422_Y64_5.MoveWork:=TRUE;	(* Förderband  Stopper Vereinzler AST/GST *)
END_ACTION

ACTION vorne_zu_action:
ST03_422_Y64_7.MoveWork:=TRUE;
END_ACTION

ACTION vorne_zu_exit:
CamResult:=0;
END_ACTION

ACTION mitte_auf_action:
ST03_422_Y64_6.MoveWork :=TRUE;
END_ACTION

ACTION Front_Cam_aktiv_exit:
RepeatCounter:=0;
CamResult:=0;
CamResult2:=0;
CamResult3:=0;
END_ACTION

ACTION Start_Front_Cam_action:
IF NOT MP.ST02.SensopartEthernet THEN
	ST03_8_80_A1.i16_job := 1;		 (*Sensopart Kamera Frontseite*)
	ST03_8_80_A1.b_start := TRUE;
ELSE
	ST03_8_90_A1.JobNo := 1;
	ST03_8_90_A1.st_ctrl_in.b_start := TRUE;
END_IF
END_ACTION

ACTION Delay_Front_Cam_entry:
IF NOT MP.ST02.SensopartEthernet THEN
	ST03_8_80_A1.b_start := FALSE;	 (*Sensopart Kamera Frontseite*)
ELSE
	ST03_8_90_A1.st_ctrl_in.b_start := FALSE;
END_IF

RepeatCounter:=RepeatCounter+1;
END_ACTION

ACTION Verarbeitet_FrontCam_entry:
IF NOT MP.ST02.SensopartEthernet THEN
	IF 	MP.ST03.FrontCamOn THEN
		IF	ST03_8_80_A1.Ergebnis_IO AND	  (*Sensopart Kamera  links*)
			NOT ST03_8_80_A1.Ergebnis_NIO THEN
			CamResult:=1;	(*   0 = noch kein Bild gemacht*)
						(*   1 =  Frontseite OK*)
						(*  11 = Frontseite und Rückseite OK*)
						(*  99 = Teil ist NOK	*)
		ELSE
			CamResult:=9;	(*   0 = noch kein Bild gemacht*)
						(*   1 =  Frontseite OK*)
						(*  11 = Frontseite und Rückseite OK*)
						(*  99 = Teil ist NOK	*)
		END_IF

	ELSE
		CamResult:=1;		(*   1 =  Frontseite OK*)
	END_IF
ELSE
		IF 	MP.ST03.FrontCamOn THEN
		IF	ST03_8_90_A1.b_Kam_Pruef_IO AND	  (*Sensopart Kamera links*)
			NOT ST03_8_90_A1.b_Kam_Pruef_NIO THEN
			CamResult:=1;	(*   0 = noch kein Bild gemacht*)
						(*   1 =  Frontseite OK*)
						(*  11 = Frontseite und Rückseite OK*)
						(*  99 = Teil ist NOK	*)
		ELSE
			CamResult:=9;	(*   0 = noch kein Bild gemacht*)
						(*   1 =  Frontseite OK*)
						(*  11 = Frontseite und Rückseite OK*)
						(*  99 = Teil ist NOK	*)
		END_IF
	
	ELSE
		CamResult:=1;		(*   1 =  Frontseite OK*)
	END_IF
END_IF
	RepeatCounter:=RepeatCounter+1;
END_ACTION

ACTION Verarbeitet_FrontCam_exit:
IF CamResult = 9 THEN
	NokCounter1li := NokCounter1li + 1;
END_IF
END_ACTION

ACTION Print_Front_OK_exit:
CamResult:=1;	(*   0 = noch kein Bild gemacht*)
			(*   1 =  Frontseite OK*)
			(*  11 = Frontseite und Rückseite OK*)
			(*  99 = Teil ist NOK	*)
END_ACTION

ACTION Back_Cam_aktiv_exit:
RepeatCounter:=0;
END_ACTION

ACTION Start_Back_Cam_action:
IF NOT MP.ST02.SensopartEthernet THEN
	ST03_8_85_A1.i16_job := 1;		 (*Sensopart Kamera rechts*)
	ST03_8_85_A1.b_start := TRUE;
ELSE
	ST03_8_95_A1.JobNo := 1;		(*Sensopart Kamera Ethernet rechts *)
	ST03_8_95_A1.st_ctrl_in.b_start := TRUE;
END_IF
END_ACTION

ACTION Delay_Back_Cam_entry:
IF NOT MP.ST02.SensopartEthernet THEN
	ST03_8_85_A1.b_start := FALSE;	 (*Sensopart Kamera rechts*)
ELSE
	ST03_8_95_A1.st_ctrl_in.b_start := FALSE;	(*Sensopart Kamera Ethernet rechts *)
END_IF

RepeatCounter:=RepeatCounter+1;
END_ACTION

ACTION Verarbeitet_BackCam_entry:
IF NOT MP.ST02.SensopartEthernet THEN
	IF 	MP.ST03.BackCamOn THEN
		IF	ST03_8_85_A1.Ergebnis_IO AND	  (*Sensopart Kamera rechts*)
			NOT ST03_8_85_A1.Ergebnis_NIO THEN
			CamResult:=CamResult+10;	(*   0 = noch kein Bild gemacht*)
							(*   1 =  Frontseite OK*)
							(*  11 = Frontseite und Rückseite OK*)
							(*  99 = Teil ist NOK	*)
		ELSE
			CamResult:=99;		(*   0 = noch kein Bild gemacht*)
							(*   1 =  Frontseite OK*)
							(*  11 = Frontseite und Rückseite OK*)
							(*  99 = Teil ist NOK	*)
		END_IF
	
	ELSE
		CamResult:=CamResult+10;		(*   1 =  Frontseite OK*)
	END_IF

ELSE
		IF 	MP.ST03.FrontCamOn THEN
		IF	ST03_8_95_A1.b_Kam_Pruef_IO AND	 (*Sensopart Kamera Ethernet rechts *)
			NOT ST03_8_95_A1.b_Kam_Pruef_NIO THEN
			CamResult:=CamResult+10;	(*   0 = noch kein Bild gemacht*)
						(*   1 =  Frontseite OK*)
						(*  11 = Frontseite und Rückseite OK*)
						(*  99 = Teil ist NOK	*)
		ELSE
			CamResult:=CamResult + 90;	(*   0 = noch kein Bild gemacht*)
						(*   1 =  Frontseite OK*)
						(*  11 = Frontseite und Rückseite OK*)
						(*  99 = Teil ist NOK	*)
		END_IF
	
	ELSE
		CamResult:=CamResult+10;		(*   1 =  Rückseite OK*)
	END_IF
END_IF
RepeatCounter:=RepeatCounter+1;
END_ACTION

ACTION Verarbeitet_BackCam_exit:
IF CamResult > 19 THEN
	NokCounter1re := NokCounter1re +1;
END_IF
END_ACTION

ACTION Print_Back_OK_exit:
CamResult:=CamResult+10;	(*   0 = noch kein Bild gemacht*)
				(*   1 =  Frontseite OK*)
				(*  11 = Frontseite und Rückseite OK*)
				(*  99 = Teil ist NOK	*)
END_ACTION

ACTION Zylinder_2_zu_action:
ST03_423_Y65_6.MoveWork := TRUE;
END_ACTION

ACTION Zylinder_1_auf_action:
ST03_422_Y64_7.MoveInit := TRUE;
END_ACTION

ACTION Front_Cam_aktiv___exit:
RepeatCounter:=0;
CamResult2:=0;
END_ACTION

ACTION Start_Front_Cam___action:
IF NOT MP.ST02.SensopartEthernet THEN
	ST03_8_80_A1.i16_job := 1;		 (*Sensopart Kamera Frontseite*)
	ST03_8_80_A1.b_start := TRUE;
ELSE
	ST03_8_90_A1.JobNo := 2;
	ST03_8_90_A1.st_ctrl_in.b_start := TRUE;
END_IF
END_ACTION

ACTION Delay_Front_Cam___entry:
IF NOT MP.ST02.SensopartEthernet THEN
	ST03_8_80_A1.b_start := FALSE;			 (*Sensopart Kamera links*)
ELSE
	ST03_8_90_A1.st_ctrl_in.b_start := FALSE;	 (*Sensopart Kamera Ethernet links *)
END_IF

RepeatCounter:=RepeatCounter+1;
END_ACTION

ACTION Verarbeitet_FrontCam___entry:
IF NOT MP.ST02.SensopartEthernet THEN
	IF 	MP.ST03.FrontCamOn THEN
		IF	ST03_8_80_A1.Ergebnis_IO AND	  (*Sensopart Kamera links*)
			NOT ST03_8_80_A1.Ergebnis_NIO THEN
			CamResult2:=1;	(*   0 = noch kein Bild gemacht*)
						(*   1 =  Frontseite OK*)
						(*  11 = Frontseite und Rückseite OK*)
						(*  99 = Teil ist NOK	*)
		ELSE
			CamResult2:=9;	(*   0 = noch kein Bild gemacht*)
						(*   1 =  Frontseite OK*)
						(*  11 = Frontseite und Rückseite OK*)
						(*  99 = Teil ist NOK	*)
		END_IF
	
	ELSE
		CamResult2:=1;		(*   1 =  Frontseite OK*)
	END_IF
ELSE
		IF 	MP.ST03.FrontCamOn THEN
		IF	ST03_8_90_A1.b_Kam_Pruef_IO AND	   (*Sensopart Kamera Ethernet links *)
			NOT ST03_8_90_A1.b_Kam_Pruef_NIO THEN
			CamResult2:=1;	(*   0 = noch kein Bild gemacht*)
						(*   1 =  Frontseite OK*)
						(*  11 = Frontseite und Rückseite OK*)
						(*  99 = Teil ist NOK	*)
		ELSE
			CamResult2:=9;	(*   0 = noch kein Bild gemacht*)
						(*   1 =  Frontseite OK*)
						(*  11 = Frontseite und Rückseite OK*)
						(*  99 = Teil ist NOK	*)
		END_IF
	
	ELSE
		CamResult2:=1;		(*   1 =  Frontseite OK*)
	END_IF
END_IF
	RepeatCounter:=RepeatCounter+1;
END_ACTION

ACTION Verarbeitet_FrontCam___exit:
IF CamResult2 = 9 THEN
	NokCounter2li := NokCounter2li +1;
END_IF
END_ACTION

ACTION Print_Front_OK___exit:
CamResult2:=1;	(*   0 = noch kein Bild gemacht*)
			(*   1 =  Frontseite OK*)
			(*  11 = Frontseite und Rückseite OK*)
			(*  99 = Teil ist NOK	*)
END_ACTION

ACTION Back_Cam_aktiv___exit:
RepeatCounter:=0;
END_ACTION

ACTION Start_Back_Cam___action:
IF NOT MP.ST02.SensopartEthernet THEN
	ST03_8_85_A1.i16_job := 1;		 (*Sensopart Kamera rechts*)
	ST03_8_85_A1.b_start := TRUE;
ELSE
	ST03_8_95_A1.JobNo := 2;		(*Sensopart Kamera Ethernet rechts *)
	ST03_8_95_A1.st_ctrl_in.b_start := TRUE;
END_IF
END_ACTION

ACTION Delay_Back_Cam___entry:
IF NOT MP.ST02.SensopartEthernet THEN
	ST03_8_85_A1.b_start := FALSE;			 (*Sensopart Kamera rechts*)
ELSE
	ST03_8_95_A1.st_ctrl_in.b_start := FALSE;	(*Sensopart Kamera Ethernet rechts *)
END_IF

RepeatCounter:=RepeatCounter+1;
END_ACTION

ACTION Verarbeitet_BackCam___entry:
IF NOT MP.ST02.SensopartEthernet THEN
	IF 	MP.ST03.BackCamOn THEN
		IF	ST03_8_85_A1.Ergebnis_IO AND	  (*Sensopart Kamera rechts*)
			NOT ST03_8_85_A1.Ergebnis_NIO THEN
			CamResult2:=CamResult2+10;	(*   0 = noch kein Bild gemacht*)
							(*   1 =  Frontseite OK*)
							(*  11 = Frontseite und Rückseite OK*)
							(*  99 = Teil ist NOK	*)
		ELSE
			CamResult2:=99;		(*   0 = noch kein Bild gemacht*)
							(*   1 =  Frontseite OK*)
							(*  11 = Frontseite und Rückseite OK*)
							(*  99 = Teil ist NOK	*)
		END_IF

	ELSE
		CamResult2:=CamResult2+10;		(*   1 =  Rückseite OK*)
	END_IF

ELSE
		IF 	MP.ST03.FrontCamOn THEN
		IF	ST03_8_95_A1.b_Kam_Pruef_IO AND	  (*Sensopart Kamera Ethernet rechts *)
			NOT ST03_8_95_A1.b_Kam_Pruef_NIO THEN
			CamResult2:=CamResult2+10;	(*   0 = noch kein Bild gemacht*)
						(*   1 =  Frontseite OK*)
						(*  11 = Frontseite und Rückseite OK*)
						(*  99 = Teil ist NOK	*)
		ELSE
			CamResult2:=CamResult2 + 90;	(*   0 = noch kein Bild gemacht*)
						(*   1 =  Frontseite OK*)
						(*  11 = Frontseite und Rückseite OK*)
						(*  99 = Teil ist NOK	*)
		END_IF

	ELSE
		CamResult2:=CamResult2+10;			(*   1 =  Rückseite OK*)
	END_IF
END_IF
RepeatCounter:=RepeatCounter+1;
END_ACTION

ACTION Verarbeitet_BackCam___exit:
IF CamResult2 > 19 THEN
	NokCounter2re := NokCounter2re +1;
END_IF
END_ACTION

ACTION Print_Back_OK___exit:
CamResult2:=CamResult2+10;	(*   0 = noch kein Bild gemacht*)
				(*   1 =  Frontseite OK*)
				(*  11 = Frontseite und Rückseite OK*)
				(*  99 = Teil ist NOK	*)
END_ACTION

ACTION Zylinder_3_zu_action:
ST03_423_Y65_7.MoveInit := TRUE;
END_ACTION

ACTION Zylinder_2_auf_action:
ST03_423_Y65_6.MoveInit := TRUE;
END_ACTION

ACTION Front_Cam_aktiv__exit:
RepeatCounter:=0;
CamResult3:=0;
END_ACTION

ACTION Start_Front_Cam__action:
IF NOT MP.ST02.SensopartEthernet THEN
	ST03_8_80_A1.i16_job := 1;		 (*Sensopart Kamera links*)
	ST03_8_80_A1.b_start := TRUE;
ELSE
	ST03_8_90_A1.JobNo := 3;		(*Sensopart Kamera Ethernet links *)
	ST03_8_90_A1.st_ctrl_in.b_start := TRUE;
END_IF
END_ACTION

ACTION Delay_Front_Cam__entry:
IF NOT MP.ST02.SensopartEthernet THEN
	ST03_8_80_A1.b_start := FALSE;	 (*Sensopart Kamera links*)
ELSE
	ST03_8_90_A1.st_ctrl_in.b_start := FALSE;	(*Sensopart Kamera Ethernet links *)
END_IF

RepeatCounter:=RepeatCounter+1;
END_ACTION

ACTION Verarbeitet_FrontCam__entry:
IF NOT MP.ST02.SensopartEthernet THEN
	IF 	MP.ST03.FrontCamOn THEN
		IF	ST03_8_80_A1.Ergebnis_IO AND	  (*Sensopart Kamera links*)
			NOT ST03_8_80_A1.Ergebnis_NIO THEN
			CamResult3:=1;	(*   0 = noch kein Bild gemacht*)
						(*   1 =  Frontseite OK*)
						(*  11 = Frontseite und Rückseite OK*)
						(*  99 = Teil ist NOK	*)
		ELSE
			CamResult3:=9;	(*   0 = noch kein Bild gemacht*)
						(*   1 =  Frontseite OK*)
						(*  11 = Frontseite und Rückseite OK*)
						(*  99 = Teil ist NOK	*)
		END_IF

	ELSE
		CamResult3:=1;		(*   1 =  Frontseite OK*)
	END_IF
ELSE
		IF 	MP.ST03.FrontCamOn THEN
		IF	ST03_8_90_A1.b_Kam_Pruef_IO AND	 (*Sensopart Kamera Ethernet links *)
			NOT ST03_8_90_A1.b_Kam_Pruef_NIO THEN
			CamResult3:=1;	(*   0 = noch kein Bild gemacht*)
						(*   1 =  Frontseite OK*)
						(*  11 = Frontseite und Rückseite OK*)
						(*  99 = Teil ist NOK	*)
		ELSE
			CamResult3:=9;	(*   0 = noch kein Bild gemacht*)
						(*   1 =  Frontseite OK*)
						(*  11 = Frontseite und Rückseite OK*)
						(*  99 = Teil ist NOK	*)
		END_IF

	ELSE
		CamResult3:=1;		(*   1 =  Frontseite OK*)
	END_IF
END_IF
	RepeatCounter:=RepeatCounter+1;
END_ACTION

ACTION Verarbeitet_FrontCam__exit:
IF CamResult3 = 9 THEN
	NokCounter3li := NokCounter3li +1;
END_IF
END_ACTION

ACTION Print_Front_OK__exit:
CamResult3:=1;	(*   0 = noch kein Bild gemacht*)
			(*   1 =  Frontseite OK*)
			(*  11 = Frontseite und Rückseite OK*)
			(*  99 = Teil ist NOK	*)
END_ACTION

ACTION Back_Cam_aktiv__exit:
RepeatCounter:=0;
END_ACTION

ACTION Start_Back_Cam__action:
IF NOT MP.ST02.SensopartEthernet THEN
	ST03_8_85_A1.i16_job := 1;		 (*Sensopart Kamera rechts*)
	ST03_8_85_A1.b_start := TRUE;
ELSE
	ST03_8_95_A1.JobNo := 3;		(*Sensopart Kamera Ethernet rechts *)
	ST03_8_95_A1.st_ctrl_in.b_start := TRUE;
END_IF
END_ACTION

ACTION Delay_Back_Cam__entry:
IF NOT MP.ST02.SensopartEthernet THEN
	ST03_8_85_A1.b_start := FALSE;	 (*Sensopart Kamera rechts*)
ELSE
	ST03_8_95_A1.st_ctrl_in.b_start := FALSE;	(*Sensopart Kamera Ethernet rechts *)
END_IF

RepeatCounter:=RepeatCounter+1;
END_ACTION

ACTION Verarbeitet_BackCam__entry:
IF NOT MP.ST02.SensopartEthernet THEN
	IF 	MP.ST03.BackCamOn THEN
		IF	ST03_8_85_A1.Ergebnis_IO AND	  (*Sensopart Kamera rechts*)
			NOT ST03_8_85_A1.Ergebnis_NIO THEN
			CamResult3:=CamResult3+10;	(*   0 = noch kein Bild gemacht*)
							(*   1 =  Frontseite OK*)
							(*  11 = Frontseite und Rückseite OK*)
							(*  99 = Teil ist NOK	*)
		ELSE
			CamResult3:= 99;		(*   0 = noch kein Bild gemacht*)
							(*   1 =  Frontseite OK*)
							(*  11 = Frontseite und Rückseite OK*)
							(*  99 = Teil ist NOK	*)
		END_IF
	
	ELSE
		CamResult3:=CamResult3+10;		(*   1 =  Frontseite OK*)
	END_IF

ELSE
		IF 	MP.ST03.BackCamOn THEN
		IF	ST03_8_95_A1.b_Kam_Pruef_IO AND	 (*Sensopart Kamera Ethernet rechts *)
			NOT ST03_8_95_A1.b_Kam_Pruef_NIO THEN
			CamResult3:=CamResult3+10;	(*   0 = noch kein Bild gemacht*)
						(*   1 =  Frontseite OK*)
						(*  11 = Frontseite und Rückseite OK*)
						(*  99 = Teil ist NOK	*)
		ELSE
			CamResult3:=CamResult3 + 90;	(*   0 = noch kein Bild gemacht*)
						(*   1 =  Frontseite OK*)
						(*  11 = Frontseite und Rückseite OK*)
						(*  99 = Teil ist NOK	*)
		END_IF
	
	ELSE
		CamResult3:=CamResult3+10;		(*   1 =  Rückseite OK*)
	END_IF
END_IF
RepeatCounter:=RepeatCounter+1;
END_ACTION

ACTION Verarbeitet_BackCam__exit:
IF CamResult3 > 19 THEN
	NokCounter3re := NokCounter3re +1;
END_IF
END_ACTION

ACTION Print_Back_OK__exit:
CamResult3:=CamResult3+10;	(*   0 = noch kein Bild gemacht*)
				(*   1 =  Frontseite OK*)
				(*  11 = Frontseite und Rückseite OK*)
				(*  99 = Teil ist NOK	*)
END_ACTION

ACTION mitte_zu__action:
ST03_422_Y64_6.MoveInit:=TRUE;
END_ACTION

ACTION hinten_auf__action:
ST03_422_Y64_5.MoveInit:=TRUE;
END_ACTION

ACTION ResetNokCounter_entry:
(*Register um eins nach hinten schieben*)
i:=0;
FOR i:=100 TO 2 BY-1 DO
   NokPercent[i] := NokPercent[i-1];
END_FOR

IF	CamResult = 11 AND
	CamResult2 = 11 AND
	CamResult3 = 11 THEN
	NokCounter:=0;
	NokPercent[1] := FALSE;
ELSIF NOT DummyTest_160pol THEN
	gNokPartsColorCam := gNokPartsColorCam+1;
	NokCounter:=NokCounter+1;
	NokPercent[1] := TRUE;
END_IF
END_ACTION

ACTION CheckCounter_entry:
(*Anzahl der Schlechtteile von den letzten 100 Prüfungen*)
i:=0;
NokCounterPercent:=0;
FOR i:=1 TO 100 BY 1 DO
  IF	NokPercent[i] THEN
	NokCounterPercent:=NokCounterPercent+1;
	END_IF
END_FOR
END_ACTION

ACTION Msg_Cam_entry:
MessageHandler.ClearMessageLines(sVisu:=Visu.Message);
END_ACTION

ACTION Msg_Cam_action:
MessageHandler.Msg.ID:='PM112';
MessageHandler.Msg.Name:='Sensopart Kam.-Erg. Prüfung  n.i.o:';
MessageHandler.Msg.Text:='Sensopart Kam.-Erg. Prüfung  n.i.o:';

MessageHandler.Msg.Color:=Color.red;
MessageHandler.Msg.Station:=3;

MessageHandler(
	Prio:=2, 								(*1=highest, .. , 4=lowest*)
	Btn1Addr:=ADR(MsgOk),				(*Address of Button1 , if Zero then Button is unvisible*)
	Btn2Addr:=0(*ADR(MsgCancel)*),			(*Address of Button2 , if Zero then Button is unvisible*)
	sVisu:=Visu.Message);
END_ACTION

ACTION Msg_Cam_exit:
MsgOk:=FALSE;
MsgCancel:=FALSE;
END_ACTION

ACTION Counter_Reset_entry:
NokCounter:=0;
(*Percent Register löschen*)
i:=0;
FOR i:=1 TO 100 BY 1 DO
  NokPercent[i]:= FALSE;
END_FOR
NokCounterPercent:=0;
END_ACTION

ACTION Msg_Cam_Percent_entry:
MessageHandler.ClearMessageLines(sVisu:=Visu.Message);
END_ACTION

ACTION Msg_Cam_Percent_action:
MessageHandler.Msg.ID:='PM113';
MessageHandler.Msg.Name:='Sensopart Kam.-Erg. Prüfung  n.i.o:';
MessageHandler.Msg.Text:='Sensopart Kam.-Erg. Prüfung n.i.o:';

MessageHandler.Msg.Color:=Color.red;
MessageHandler.Msg.Station:=3;

MessageHandler(
	Prio:=2, 								(*1=highest, .. , 4=lowest*)
	Btn1Addr:=ADR(MsgOk),				(*Address of Button1 , if Zero then Button is unvisible*)
	Btn2Addr:=0(*ADR(MsgCancel)*),			(*Address of Button2 , if Zero then Button is unvisible*)
	sVisu:=Visu.Message);
END_ACTION

ACTION Msg_Cam_Percent_exit:
MsgOk:=FALSE;
MsgCancel:=FALSE;
END_ACTION

ACTION Zylinder_3_auf__action:
ST03_423_Y65_7.MoveWork := TRUE;
END_ACTION

ACTION Zylinder_3_auf__exit:
(*Ergebnis Protduktion*)
Result160pol:=CamResult;

IF	CamResult =11 AND
	CamResult2 = 11 AND
	CamResult3 = 11 THEN
	ST03_Main.Result:=RESULT_OK;
ELSE
	ST03_Main.Result:=RESULT_NOK;
END_IF
END_ACTION

ACTION Zylinder_1_zu__action:
ST03_422_Y64_7.MoveWork:=TRUE;
END_ACTION

ACTION SeqEnd_action:
SFCTime:=TIME_TO_DINT(TIME()-SFCTimeStart);
State:=STATE_WAIT;
END_ACTION

TRANSITION OK:
NOT MP.ST03.SGM_3621
OR
ST03_S18.BitInToCheck
END_TRANSITION

TRANSITION OK:
(
ST03_70U3_1.BitInToCheck	 AND	 	(*Bereit/ Im Druck Tintenstrahldrucker Frontseite*)
ST03_71U3_1.BitInToCheck	 AND		 (*Bereit/ Im Druck Tintenstrahldrucker Rückseite*)
NOT ST03_70U3_3.BitInToCheck AND	 (*Fehler/Störung Tintenstrahldrucker Frontseite*)
NOT ST03_71U3_3.BitInToCheck AND	 (*Fehler/Störung Tintenstrahldrucker Rückseite*)
ST03_70U3_2.BitInToCheck AND 		(*Tank voll Tintenstrahldrucker Frontseite*)
ST03_71U3_2.BitInToCheck  			(*Tank voll Tintenstrahldrucker Rückseite*)
) OR
(*b_Printer_Off OR*)
DummyTest_160pol
OR
( MP.ST03.SGM_3621 AND
ST03_70U3_1.BitInToCheck	 AND	 	(*Bereit/ Im Druck Tintenstrahldrucker Frontseite*)
ST03_71U3_1.BitInToCheck	 AND		 (*Bereit/ Im Druck Tintenstrahldrucker Rückseite*)
NOT ST03_70U3_3.BitInToCheck AND	 (*Fehler/Störung Tintenstrahldrucker Frontseite*)
NOT ST03_71U3_3.BitInToCheck )	 (*Fehler/Störung Tintenstrahldrucker Rückseite*)
END_TRANSITION

TRANSITION Front_NOK:
NOT ST03_70U3_1.BitInToCheck	  (*Bereit/ Im Druck Tintenstrahldrucker Frontseite*)
END_TRANSITION

TRANSITION Back_NOK:
NOT ST03_71U3_1.BitInToCheck	  (*Bereit/ Im Druck Tintenstrahldrucker Rückseite*)
END_TRANSITION

TRANSITION TankFront_leer:
NOT MP.ST03.SGM_3621 AND
NOT ST03_70U3_2.BitInToCheck  	(*Tank voll Tintenstrahldrucker Frontseite*)
END_TRANSITION

TRANSITION TankBack_leer:
NOT MP.ST03.SGM_3621 AND
NOT ST03_71U3_2.BitInToCheck  	(*Tank voll Tintenstrahldrucker Rückseite*)
END_TRANSITION

TRANSITION ErrFront:
ST03_70U3_3.BitInToCheck  (*Fehler/Störung Tintenstrahldrucker Frontseite*)
END_TRANSITION

TRANSITION ErrBack:
ST03_71U3_3.BitInToCheck  (*Fehler/Störung Tintenstrahldrucker Rückseite*)
END_TRANSITION

TRANSITION Frontcam_bb:
NOT MP.ST03.FrontCamOn OR
(NOT ST03_8_80_A1.b_kamera_aktiv		 (*Sensopart Kamera Frontseite*)
AND
NOT ST03_8_80_A1.sm_kamera_nicht_bb  (*Sensopart Kamera Frontseite*)
AND
NOT ST03_8_90_A1.sm_kamera_nicht_bb
AND
ST03_8_90_A1.st_ctrl_out.b_bereit
AND
ST03_8_90_A1.Activated)
END_TRANSITION

TRANSITION Backcam_bb:
NOT MP.ST03.BackCamOn OR
(NOT ST03_8_85_A1.b_kamera_aktiv		 (*Sensopart Kamera rechts*)
AND
NOT ST03_8_85_A1.sm_kamera_nicht_bb	 (*Sensopart Kamera rechts*)
AND
NOT ST03_8_95_A1.sm_kamera_nicht_bb	(*Sensopart Kamera Ethernet rechts *)
AND
ST03_8_95_A1.st_ctrl_out.b_bereit			(*Sensopart Kamera Ethernet rechts *)
AND
ST03_8_95_A1.Activated)
END_TRANSITION

TRANSITION Vereinzler_frei:
NOT ST03_421_B63_7.BitInToCheck 			(*  ISK anwesend am Vereinzler*)
END_TRANSITION

TRANSITION StateOk:
ST03_422_Y64_5.State=STATE_OK AND
ST03_422_Y64_6.State=STATE_OK AND
ST03_421_B63_7.BitInToCheck 			(*  ISK anwesend am Vereinzler*)
AND
gTipImp
END_TRANSITION

TRANSITION StateOk:
ST03_422_Y64_5.State=STATE_OK
AND
gTipImp
END_TRANSITION

TRANSITION Print_Cam_free:
NOT ST03_422_B64_3.BitInToCheck	 AND	(* Förderband ISK anwesend Stopper 1 Kamera*)
NOT ST03_423_B65_2.BitInToCheck	AND (* Förderband ISK anwesend Stopper Kamera 2*)
NOT ST03_423_B65_5.BitInToCheck	AND (* Förderband ISK anwesend Stopper 3 Kamera*)
NOT ST03_422_B64_0.BitInToCheck	AND(* Förderband Trigger Tintenstrahldrucker (Lichtschranke 1)*)
NOT ST03_423_B66_0.BitInToCheck	(* Förderband Trigger Tintenstrahldrucker (Lichtschranke 2)*)
AND
gTipImp
END_TRANSITION

TRANSITION StateOk:
ST03_422_Y64_7.State=STATE_OK AND
ST03_422_Y64_6.State=STATE_OK AND
gTipImp
END_TRANSITION

TRANSITION Iso_on_CamPos:
ST03_422_B64_3.BitInToCheck	 (* Förderband ISK anwesend Stopper 1 Kamera*)
AND
gTipImp
END_TRANSITION

TRANSITION aktiv:
ST03_8_80_A1.b_kamera_aktiv OR(*Sensopart Kamera Frontseite*)
ST03_8_90_A1.Activated
END_TRANSITION

TRANSITION Busy:
ST03_8_80_A1.b_busy OR  (*Sensopart Kamera Frontseite*)
ST03_8_90_A1.st_ctrl_out.b_busy
END_TRANSITION

TRANSITION Done:
(ST03_8_80_A1.b_done AND	 (*Sensopart Kamera Frontseite*)(
(ST03_8_80_A1.Ergebnis_IO AND NOT ST03_8_80_A1.Ergebnis_NIO)OR
RepeatCounter>=2 ))
OR
(ST03_8_90_A1.st_ctrl_out.b_fertig AND
((ST03_8_90_A1.b_Kam_Pruef_IO AND NOT ST03_8_90_A1.b_Kam_Pruef_NIO) OR
RepeatCounter>=2))
END_TRANSITION

TRANSITION CamNotAktiv:
(ST03_8_80_A1.b_done	 (*Sensopart Kamera Frontseite*)
AND
NOT MP.ST03.FrontCamOn)
OR
(ST03_8_90_A1.st_ctrl_out.b_fertig  (*Kamera Farberkennung Ethernet*)
AND
NOT MP.ST03.FrontCamOn)
END_TRANSITION

TRANSITION CamDone:
ST03_8_80_A1.b_done	 (*Sensopart Kamera links*)
OR
ST03_8_90_A1.st_ctrl_out.b_fertig	 (*Sensopart Kamera Ethernet links *)
END_TRANSITION

TRANSITION aktiv:
ST03_8_85_A1.b_kamera_aktiv OR 	(*Sensopart Kamera rechts*)
ST03_8_95_A1.Activated			(*Sensopart Kamera Ethernet rechts *)
END_TRANSITION

TRANSITION Busy:
ST03_8_85_A1.b_busy OR				 (*Sensopart Kamera rechts*)
ST03_8_95_A1.st_ctrl_out.b_busy		(*Sensopart Kamera Ethernet rechts *)
END_TRANSITION

TRANSITION Done:
(ST03_8_85_A1.b_done AND		 (*Sensopart Kamera rechts*)
((ST03_8_85_A1.Ergebnis_IO AND NOT ST03_8_85_A1.Ergebnis_NIO)OR
RepeatCounter>=2 ))
OR
(ST03_8_95_A1.st_ctrl_out.b_fertig AND	(*Sensopart Kamera Ethernet rechts *)
((ST03_8_95_A1.b_Kam_Pruef_IO AND NOT ST03_8_95_A1.b_Kam_Pruef_NIO) OR
RepeatCounter>=2))
END_TRANSITION

TRANSITION CamNotAktiv:
(ST03_8_85_A1.b_done				 (*Sensopart Kamera rechts*)
AND
NOT MP.ST03.BackCamOn)
OR
(ST03_8_95_A1.st_ctrl_out.b_fertig 	(*Sensopart Kamera Ethernet rechts *)
AND
NOT MP.ST03.BackCamOn)
END_TRANSITION

TRANSITION CamDone:
ST03_8_85_A1.b_done				 (*Sensopart Kamera rechts*)
OR
ST03_8_95_A1.st_ctrl_out.b_fertig	(*Sensopart Kamera Ethernet rechts *)
END_TRANSITION

TRANSITION StateOk:
ST03_423_Y65_6.State = STATE_OK AND
gTipImp
END_TRANSITION

TRANSITION StateOk:
ST03_422_Y64_7.State = STATE_OK AND
gTipImp
END_TRANSITION

TRANSITION Iso_on_CamPos_2:
ST03_423_B65_2.BitInToCheck	 (* Förderband ISK anwesend Stopper Kamera*)
AND
gTipImp
END_TRANSITION

TRANSITION aktiv:
ST03_8_80_A1.b_kamera_aktiv OR(*Sensopart Kamera Frontseite*)
ST03_8_90_A1.Activated
END_TRANSITION

TRANSITION Busy:
ST03_8_80_A1.b_busy OR  			(*Sensopart Kamera links*)
ST03_8_90_A1.st_ctrl_out.b_busy	 (*Sensopart Kamera Ethernet links *)
END_TRANSITION

TRANSITION Done:
(ST03_8_80_A1.b_done AND		 (*Sensopart Kamera links*)
(
(ST03_8_80_A1.Ergebnis_IO AND NOT ST03_8_80_A1.Ergebnis_NIO)OR
RepeatCounter>=2 ))
OR

(ST03_8_90_A1.st_ctrl_out.b_fertig AND		 (*Sensopart Kamera Ethernet links *)
((ST03_8_90_A1.b_Kam_Pruef_IO AND NOT ST03_8_90_A1.b_Kam_Pruef_NIO) OR
RepeatCounter>=2))
END_TRANSITION

TRANSITION CamNotAktiv:
(ST03_8_80_A1.b_done	 (*Sensopart Kamera links*)
AND
NOT MP.ST03.FrontCamOn)
OR
(ST03_8_90_A1.st_ctrl_out.b_fertig   (*Sensopart Kamera Ethernet links *)
AND
NOT MP.ST03.FrontCamOn)
END_TRANSITION

TRANSITION CamDone:
ST03_8_80_A1.b_done	 (*Sensopart Kamera links*)
OR
ST03_8_90_A1.st_ctrl_out.b_fertig	(*Sensopart Kamera Ethernet links *)
END_TRANSITION

TRANSITION aktiv:
ST03_8_85_A1.b_kamera_aktiv OR 	(*Sensopart Kamera rechts*)
ST03_8_95_A1.Activated			(*Sensopart Kamera Ethernet rechts *)
END_TRANSITION

TRANSITION Busy:
ST03_8_85_A1.b_busy OR			 (*Sensopart Kamera rechts*)
ST03_8_95_A1.st_ctrl_out.b_busy	(*Sensopart Kamera Ethernet rechts *)
END_TRANSITION

TRANSITION Done:
(ST03_8_85_A1.b_done AND				 (*Sensopart Kamera rechts*)
((ST03_8_85_A1.Ergebnis_IO AND NOT ST03_8_85_A1.Ergebnis_NIO)OR
RepeatCounter>=2 ))
OR
(ST03_8_95_A1.st_ctrl_out.b_fertig AND		(*Sensopart Kamera Ethernet rechts *)
((ST03_8_95_A1.b_Kam_Pruef_IO AND NOT ST03_8_95_A1.b_Kam_Pruef_NIO) OR
RepeatCounter>=2))
END_TRANSITION

TRANSITION CamNotAktiv:
(ST03_8_85_A1.b_done	 			(*Sensopart Kamera rechts*)
AND
NOT MP.ST03.BackCamOn)
OR
(ST03_8_95_A1.st_ctrl_out.b_fertig 	(*Sensopart Kamera Ethernet rechts *)
AND
NOT MP.ST03.BackCamOn)
END_TRANSITION

TRANSITION CamDone:
ST03_8_85_A1.b_done				 (*Sensopart Kamera rechts*)
OR
ST03_8_95_A1.st_ctrl_out.b_fertig	 (*Sensopart Kamera Ethernet rechts *)
END_TRANSITION

TRANSITION StateOk:
ST03_423_Y65_7.State = STATE_OK AND
gTipImp
END_TRANSITION

TRANSITION StateOk:
ST03_423_Y65_6.State = STATE_OK AND
gTipImp
END_TRANSITION

TRANSITION Iso_on_CamPos_2:
ST03_423_B65_5.BitInToCheck	 (* Förderband ISK anwesend Stopper Kamera*)
AND
gTipImp
END_TRANSITION

TRANSITION aktiv:
ST03_8_80_A1.b_kamera_aktiv OR	(*Sensopart Kamera links*)
ST03_8_90_A1.Activated			(*Sensopart Kamera Ethernet links *)
END_TRANSITION

TRANSITION Busy:
ST03_8_80_A1.b_busy OR 			 (*Sensopart Kamera links*)
ST03_8_90_A1.st_ctrl_out.b_busy	(*Sensopart Kamera Ethernet links *)
END_TRANSITION

TRANSITION Done:
(ST03_8_80_A1.b_done AND	 (*Sensopart Kamera links*)
(
(ST03_8_80_A1.Ergebnis_IO AND NOT ST03_8_80_A1.Ergebnis_NIO)OR
RepeatCounter>=2 ))
OR
(ST03_8_90_A1.st_ctrl_out.b_fertig AND	(*Sensopart Kamera Ethernet links *)
((ST03_8_90_A1.b_Kam_Pruef_IO AND NOT ST03_8_90_A1.b_Kam_Pruef_NIO) OR
RepeatCounter>=2))
END_TRANSITION

TRANSITION CamNotAktiv:
(ST03_8_80_A1.b_done	 (*Sensopart Kamera links*)
AND
NOT MP.ST03.FrontCamOn)
OR
(ST03_8_90_A1.st_ctrl_out.b_fertig  (*Sensopart Kamera Ethernet links *)
AND
NOT MP.ST03.FrontCamOn)
END_TRANSITION

TRANSITION CamDone:
ST03_8_80_A1.b_done				 (*Sensopart Kamera links*)
OR
ST03_8_90_A1.st_ctrl_out.b_fertig	 (*Sensopart Kamera Ethernet links *)
END_TRANSITION

TRANSITION aktiv:
ST03_8_85_A1.b_kamera_aktiv OR		 (*Sensopart Kamera rechts*)
ST03_8_95_A1.Activated				(*Sensopart Kamera Ethernet rechts *)
END_TRANSITION

TRANSITION Busy:
ST03_8_85_A1.b_busy OR			 (*Sensopart Kamera rechts*)
ST03_8_95_A1.st_ctrl_out.b_busy	(*Sensopart Kamera Ethernet rechts *)
END_TRANSITION

TRANSITION Done:
(ST03_8_85_A1.b_done AND				 (*Sensopart Kamera rechts*)
((ST03_8_85_A1.Ergebnis_IO AND NOT ST03_8_85_A1.Ergebnis_NIO)OR
RepeatCounter>=2 ))
OR
(ST03_8_95_A1.st_ctrl_out.b_fertig AND		(*Sensopart Kamera Ethernet rechts *)
((ST03_8_95_A1.b_Kam_Pruef_IO AND NOT ST03_8_95_A1.b_Kam_Pruef_NIO) OR
RepeatCounter>=2))
END_TRANSITION

TRANSITION CamNotAktiv:
(ST03_8_85_A1.b_done	 			(*Sensopart Kamera rechts*)
AND
NOT MP.ST03.BackCamOn)
OR
(ST03_8_95_A1.st_ctrl_out.b_fertig  (*Sensopart Kamera Ethernet rechts *)
AND
NOT MP.ST03.BackCamOn)
END_TRANSITION

TRANSITION CamDone:
ST03_8_85_A1.b_done	 			(*Sensopart Kamera rechts*)
OR
ST03_8_95_A1.st_ctrl_out.b_fertig	 (*Sensopart Kamera Ethernet rechts *)
END_TRANSITION

TRANSITION StateOk:
ST03_422_Y64_6.State=STATE_OK AND
gTipImp
END_TRANSITION

TRANSITION StateOk:
ST03_422_Y64_5.State=STATE_OK AND
gTipImp
END_TRANSITION

TRANSITION CounterOK:
NokCounter<MP.ST03.CamNoOfErrors AND
NokCounterPercent < MP.ST03.CamNoOfErrorsPercent
END_TRANSITION

TRANSITION Nok_Cont:
NokCounter >= MP.ST03.CamNoOfErrors
END_TRANSITION

TRANSITION Nok_Percent:
NokCounterPercent >= MP.ST03.CamNoOfErrorsPercent
END_TRANSITION

TRANSITION Cam_full:
ST03_423_B65_5.BitInToCheck  (* Förderband ISK anwesend Stopper 3 Kamera*)
END_TRANSITION

TRANSITION free:
NOT ST03_422_B64_4.BitInToCheck AND		(* Zuführung ISK auf Übergabeposition Robo Palettierer*)
ST03_423_B65_5.BitInToCheck		AND			(* Förderband ISK anwesend Stopper Kamera*)
Robot01.ActualArea <> 4
END_TRANSITION

TRANSITION StateOk:
ST03_423_Y65_7.State = STATE_OK AND
ST03_422_B64_4.BitInToCheck AND		(* Zuführung ISK auf Übergabeposition Robo Palettierer*)
NOT ST03_423_B65_5.BitInToCheck		(* Förderband ISK anwesend Stopper Kamera*)
AND
gTipImp
END_TRANSITION

TRANSITION StateOk:
ST03_422_Y64_7.State=STATE_OK
AND
gTipImp
END_TRANSITION
END_PROGRAM

(* POU Stations/ST_03_Ruestsaetze/ST_03_PRGs/ST03_Autostop, ST *)
PROGRAM ST03_Autostop
VAR_INPUT
	Start										:BOOL;
END_VAR
VAR_OUTPUT
END_VAR

VAR
	fb_ton_Autostop						: TON;
	fb_r_trig_Autostop					: R_TRIG;
	Error								: BOOL;
	MsgOK								: BOOL;
END_VAR
fb_ton_Autostop(IN:=Start, PT:=t#500m );
IF	MP.ST00.Override > 0 THEN
	fb_ton_Autostop.PT:=fb_ton_Autostop.PT * (100 / MP.ST00.Override) ;
END_IF

fb_r_trig_Autostop(CLK:=fb_ton_Autostop.Q);
IF	fb_r_trig_Autostop.Q AND
	(gTypeCode=312 OR		 (*nur beim 93 pol*)
	 gTypeCode=4991) THEN 	(*nur beim 102 pol*)
	ModeSelect.iRemoteAutoStop:=TRUE;
	Start:=FALSE;
	Error:=TRUE;
	MessageHandler.ClearMessageLines(sVisu:=Visu.Message);

END_IF

IF	Error THEN
	MessageHandler.Msg.ID:='PM20';
	MessageHandler.Msg.Name:='Timeout';
	MessageHandler.Msg.Text:='Autostop weil die Anlage zu lange gestanden ist!' ;
	MessageHandler.Msg.Color:=Color.yellow;
	MessageHandler.Msg.Station:=0;

	MessageHandler(
		Prio:=2, 							(*1=highest, .. , 4=lowest*)
		Btn1Addr:=ADR(MsgOk),			(*Address of Button1 , if Zero then Button is unvisible*)
		Btn2Addr:=,						(*Address of Button2 , if Zero then Button is unvisible*)
		sVisu:=Visu.Message);

	IF 	MsgOK THEN
		MsgOk:=FALSE;
		Error:=FALSE;
	END_IF

END_IF
END_PROGRAM

(* POU Stations/ST_03_Ruestsaetze/ST_03_PRGs/ST03_Init_AbholPos, ST *)
PROGRAM ST03_Init_AbholPos
VAR
	RoboPos31		:BOOL;
	RoboPos35		:BOOL;
	RoboPosErr		:BOOL;
	CamDone			:BOOL;
	fb_Ton_PosErr	:TON;

	MsgOK			: BOOL;
END_VAR
(* Hier werden alle Abholpositionen am Rüstsatz bestimmt.
Ausnahmen:
	alte Rüstsätze:
		P360 74pol 
		P379 91pol 
		P489 168pol
		P4992 35pol
	Tampondrucker:
		P312 93pol
		P4991 102pol			*)

RoboPos31:=FALSE;
RoboPos35:=FALSE;
RoboPosErr:=FALSE;
CASE  gTypeCode OF

360,489:	(*74polig, 91polig, 168polig*)

	RoboPos31:=TRUE;

379: (*91 pol*)
RoboPos31:=
		ST08_412_B59_0.BitInToCheck;
	ST03_Main.Result:=RESULT_OK;		(* immer OK, wenn es keine Prüfung gibt*)

4992: (*35polig*)
	RoboPos31:=
		NOT ST08_412_B58_5_35pol.BitInToCheck AND	(*links*)
		ST08_412_B58_6_35pol.BitInToCheck;			(*rechts*)
	RoboPos35:=
		ST08_412_B58_5_35pol.BitInToCheck AND		(*links*)
		NOT ST08_412_B58_6_35pol.BitInToCheck;		(*rechts*)
	RoboPosErr:=
		ST08_412_B58_5_35pol.BitInToCheck AND		(*links*)
		ST08_412_B58_6_35pol.BitInToCheck;			(*rechts*)
	ST03_Main.Result:=RESULT_OK;		(* immer OK, wenn es keine Prüfung gibt*)

4871:(*154polig*)
	RoboPos31:=
		ST03_426_B68_4.BitInToCheck; 		(* Zuführung ISK auf Übergabeposition Robo Palettierer*)
	ST03_Main.Result:=RESULT_OK;		(* immer OK, wenn es keine Prüfung gibt*)

4872:(*154 Rasterplatte*)
	RoboPos31:=
			ST03_419_B61_2.BitInToCheck AND 	(*  Züführung links ISK auf Übergabeposition Roboter Palettierer*)
			ST03_419_B61_3.BitInToCheck;		(*  Züführung rechts ISK auf Übergabeposition Roboter Palettierer*)
	ST03_Main.Result:=RESULT_OK;			(* immer OK, wenn es keine Prüfung gibt*)

322: (*160polig*)
	RoboPos31:=
		ST03_422_B64_4.BitInToCheck; 			(* Zuführung ISK auf Übergabeposition Robo Palettierer*)

522:(*P522 206 polig*)
	RoboPos31:=
		ST03_437_B68_4.BitInToCheck AND
		NOT ST03_436_B68_1.BitInToCheck AND	(*links*)
		ST03_436_B68_2.BitInToCheck;			(*rechts*)
	RoboPos35:=
		ST03_437_B68_4.BitInToCheck AND
		ST03_436_B68_1.BitInToCheck AND		(*links*)
		NOT ST03_436_B68_2.BitInToCheck;		(*rechts*)
	RoboPosErr:=
(*		ST03_437_B68_4.BitInToCheck AND*)
		ST03_436_B68_1.BitInToCheck AND		(*links*)
		ST03_436_B68_2.BitInToCheck;		(*rechts*)
	ST03_Main.Result:=RESULT_OK;		(* immer OK, wenn es keine Prüfung gibt*)

550:(*P550 92 polig*)
	RoboPos31:=
		ST03_446_B70_4.BitInToCheck AND
		ST03_445_B70_1.BitInToCheck	AND		(*rechts*)
		NOT ST03_445_B70_2.BitInToCheck;			(*links*)
	RoboPos35:=
		ST03_446_B70_4.BitInToCheck AND
		NOT ST03_445_B70_1.BitInToCheck	AND	(*rechts*)
		ST03_445_B70_2.BitInToCheck;				(*links*)
	RoboPosErr:=
		ST03_446_B70_4.BitInToCheck AND
		ST03_445_B70_1.BitInToCheck AND	(*links*)
		ST03_445_B70_2.BitInToCheck;		(*rechts*)
	ST03_Main.Result:=RESULT_OK;		(* immer OK, wenn es keine Prüfung gibt*)

564:(*P564 124 polig*)
	RoboPos31:=
		ST03_453_B70_4.BitInToCheck AND
		ST03_452_B70_1.BitInToCheck	AND	(*rechts*)
		NOT	ST03_452_B70_2.BitInToCheck;	(*links*)
	RoboPos35:=
		ST03_453_B70_4.BitInToCheck AND
		NOT ST03_452_B70_1.BitInToCheck	AND	(*rechts*)
		ST03_452_B70_2.BitInToCheck;				(*links*)
	RoboPosErr:=
		ST03_446_B70_4.BitInToCheck AND
		ST03_445_B70_1.BitInToCheck AND	(*links*)
		ST03_445_B70_2.BitInToCheck;		(*rechts*)
	ST03_Main.Result:=RESULT_OK;		(* immer OK, wenn es keine Prüfung gibt*)

569:(*P569 46 polig*)
	RoboPos31:=
		ST03_463_B70_7.BitInToCheck AND
		ST03_462_B70_1.BitInToCheck	AND	(*rechts*)
		NOT	ST03_462_B70_2.BitInToCheck;	(*links*)
	RoboPos35:=
		ST03_463_B70_7.BitInToCheck AND
		NOT ST03_462_B70_1.BitInToCheck	AND(*rechts*)
		ST03_462_B70_2.BitInToCheck;
	RoboPosErr:=
		ST03_463_B70_7.BitInToCheck AND
		ST03_462_B70_1.BitInToCheck AND 	(*links*)
		ST03_462_B70_2.BitInToCheck;		(*rechts*)
	ST03_Main.Result:=RESULT_OK;		(* immer OK, wenn es keine Prüfung gibt*)

5731:(*P573 88polig*)
	RoboPos31:=
		ST03_501_B69_7. BitInToCheck AND	(*ISK auf Abholposition Robi*)
		NOT ST03_502_B70_0.BitInToCheck;	(*ISK Lageerkennung*)
	RoboPos35:=
		ST03_501_B69_7. BitInToCheck AND	(*ISK auf Abholposition Robi*)
		ST03_502_B70_0.BitInToCheck;		(*ISK Lageerkennung*)
	ST03_Main.Result:=RESULT_OK;		(* immer OK, wenn es keine Prüfung gibt*)

575,5753,5754,5755:(*P575 7polig*)
	RoboPos31:=
		ST03_513_B70_7.BitInToCheck AND		(*ISK auf Übergabeposition  1*)
		ST03_514_B71_2.BitInToCheck	AND	(*ISK auf Übergabeposition  2*)
		ST03_514_B71_5.BitInToCheck	AND	(*ISK auf Übergabeposition  3*)
		ST03_514_B71_6.BitInToCheck;			(*ISK auf Übergabeposition  4*)
	ST03_Main.Result:=RESULT_OK;			(* immer OK, wenn es keine Prüfung gibt*)

5732:(*P573 88polig AMG*)
	RoboPos31:=
		ST03_521_B69_7. BitInToCheck AND	(*ISK Lageerkennung links*)
		NOT ST03_522_B70_0.BitInToCheck;	(*ISK Lageerkennung rechts*)
	RoboPos35:=
		NOT ST03_521_B69_7. BitInToCheck AND(*ISK Lageerkennung links*)
		ST03_522_B70_0.BitInToCheck;			(*ISK Lageerkennung rechts*)
	RoboPosErr:=
		ST03_521_B69_7.BitInToCheck AND	(*links*)
		ST03_522_B70_0.BitInToCheck;		(*rechts*)
	ST03_Main.Result:=RESULT_OK;		(*immer OK, wenn es keine Prüfung gibt*)

5631:(*NOX 4pol*)
	RoboPos31:=
		ST03_491_B69_7.BitInToCheck;		(*Zuführung ISK auf Übergabeposition Robo Palettierer*)
	ST03_Main.Result:=RESULT_OK;		(*immer OK, wenn es keine Prüfung gibt*)

5632:(*NOX 5pol*)
	RoboPos31:=
		ST03_4x3_B70_0.BitInToCheck AND 	(*Pos 1*)		(* ISK anwesend Übergabeposition Stopper *)
		ST03_4x3_B70_1.BitInToCheck; (*AND	(*Pos 2*)		(* ISK anwesend Übergabeposition *)
		ST03_NOX_5pol_Zufuehrung.Result <> RESULT_NON; *)	(*warte bis Kamera fertig ist*)
	ST03_Main.Result:=ST03_NOX_5pol_Zufuehrung.Result;

5633:(*NOX 6pol*)
	RoboPos31:=
		ST03_4x3_B70_0.BitInToCheck AND 	(*Pos 1*)		(* ISK anwesend Übergabeposition Stopper *)
		ST03_4x3_B70_1.BitInToCheck AND	(*Pos 2*)		(* ISK anwesend Übergabeposition *)
		NOT ST03_NOX_6pol_Zufuehrung.LockForCam; 		(*warte bis Kamera fertig ist*)
	ST03_Main.Result:=ST03_NOX_6pol_Zufuehrung.Result;

5771:(*P5771 120polig*);
	RoboPos31:=
		ST03_531_B69_7. BitInToCheck AND	(*ISK rechts Lageerkennung*)
		NOT ST03_532_B70_0.BitInToCheck;	(*ISK links Lageerkennung*)
	RoboPos35:=
		NOT ST03_531_B69_7. BitInToCheck AND	(*ISK rechts Lageerkennung*)
		ST03_532_B70_0.BitInToCheck;		(*ISK links Lageerkennung*)
	RoboPosErr:=
		ST03_531_B69_7.BitInToCheck AND	(*links*)
		ST03_532_B70_0.BitInToCheck;		(*rechts*)

	ST03_Main.Result:=RESULT_OK;		(*immer OK, wenn es keine Prüfung gibt*)

5772:(*P5772 21polig*)
	RoboPos31:=
		NOT ST03_536_B69_7. BitInToCheck AND	(*ISK anwesend an Abholposition*)
		ST03_537_B70_0.BitInToCheck;	(*ISK Lageerkennung*)
	RoboPos35:=
		ST03_536_B69_7. BitInToCheck AND	(*ISK anwesend an Abholposition*)
		ST03_537_B70_0.BitInToCheck;		(*ISK Lageerkennung*)
	RoboPosErr:=
		ST03_536_B69_7.BitInToCheck AND			(*links*)
		NOT ST03_537_B70_0.BitInToCheck;		(*rechts*)
	ST03_Main.Result:=RESULT_OK;		(*immer OK, wenn es keine Prüfung gibt*)

580:(*P580 191polig*)
	RoboPos31:=
		ST03_541_B69_7. BitInToCheck AND		(*ISK links Lageerkennung*)
		NOT ST03_542_B70_0.BitInToCheck;		(*ISK rechts Lageerkennung*)
	RoboPos35:=
		NOT ST03_541_B69_7. BitInToCheck AND	(*ISK links Lageerkennung*)
		ST03_542_B70_0.BitInToCheck;				(*ISK rechts Lageerkennung*)
	RoboPosErr:=
		ST03_541_B69_7.BitInToCheck AND	(*links*)
		ST03_542_B70_0.BitInToCheck;		(*rechts*)
	ST03_Main.Result:=RESULT_OK;		(*immer OK, wenn es keine Prüfung gibt*)

5831:(*P5831 72polig*)
	RoboPos31:=
		ST03_546_B69_7. BitInToCheck AND		(*ISK rechts Lageerkennung*)
		NOT ST03_547_B70_0.BitInToCheck;		(*ISK links Lageerkennung*)
	RoboPos35:=
		NOT ST03_546_B69_7. BitInToCheck AND	(*ISK rechts Lageerkennung*)
		ST03_547_B70_0.BitInToCheck;				(*ISK links Lageerkennung*)
	RoboPosErr:=
		ST03_546_B69_7.BitInToCheck AND	(*links*)
		ST03_547_B70_0.BitInToCheck;		(*rechts*)
	ST03_Main.Result:=RESULT_OK;		(*immer OK, wenn es keine Prüfung gibt*)

5832:(*P5832 48polig*)
	RoboPos31:=
		ST03_551_B69_7. BitInToCheck AND		(*ISK rechts Lageerkennung*)
		NOT ST03_552_B70_0.BitInToCheck;		(*ISK links Lageerkennung*)
	RoboPos35:=
		NOT ST03_551_B69_7. BitInToCheck AND	(*ISK rechts Lageerkennung*)
		ST03_552_B70_0.BitInToCheck;				(*ISK links Lageerkennung*)
	RoboPosErr:=
		ST03_551_B69_7.BitInToCheck AND	(*links*)
		ST03_552_B70_0.BitInToCheck;		(*rechts*)
	ST03_Main.Result:=RESULT_OK;		(*immer OK, wenn es keine Prüfung gibt*)

5841, 4993:(*P5841 268pol, 102pol neu*)

	RoboPos31:=
		ST03_556_B69_7. BitInToCheck;		(*ISK anwesend an Abholposition*)

	ST03_Main.Result:=RESULT_OK;		(*immer OK, wenn es keine Prüfung gibt*)

5842:(*P584 268poligRP*)
	RoboPos31:=
	ST03_562_B67_7. BitInToCheck AND		(*Zuführung 1 ISK auf Übergabepos. Robi*)
	ST03_563_B70_7. BitInToCheck;			(*Zuführung 2 ISK auf Übergabepos. Robi*)
	ST03_Main.Result:=RESULT_OK;		(*immer OK, wenn es keine Prüfung gibt*)

598:(*P598 33polig*)

	RoboPos31:=
		ST03_571_B69_7. BitInToCheck;		(*ISK anwesend an Abholposition*)

	ST03_Main.Result:=RESULT_OK;		(*immer OK, wenn es keine Prüfung gibt*)

END_CASE

IF	RoboPos31 AND RoboPos35 THEN
	RoboPos31:=FALSE;
	RoboPos35:=FALSE;
END_IF


fb_Ton_PosErr(IN:=RoboPosErr,PT:=t#1s);
IF	ModeSelect.Mode>MODE_MANUAL AND fb_Ton_PosErr.Q THEN

	IF 	MessageHandler.Msg.ID <> 'PM122' THEN
		MessageHandler.ClearMessageLines(sVisu:=Visu.Message);
	END_IF
	MessageHandler.Msg.ID:='PM122';
	MessageHandler.Msg.Name:='Zuführung Lageerkennung';
	MessageHandler.Msg.Text:='Zuführung Lageerkennung prüfen';
	MessageHandler.Msg.Color:=Color.red;
	MessageHandler.Msg.Station:=0;

	MessageHandler(
		Prio:=2, 						(*1=highest, .. , 4=lowest*)
		Btn1Addr:=ADR(MsgOk),		(*Address of Button1 , if Zero then Button is unvisible*)
		Btn2Addr:=,					(*Address of Button2 , if Zero then Button is unvisible*)
		sVisu:=Visu.Message);

	IF 	MsgOK  OR NOT fb_Ton_PosErr.Q THEN
		MsgOk:=FALSE;
	END_IF

END_IF
END_PROGRAM

(* POU Stations/ST_03_Ruestsaetze/ST_03_SFCs/Zufuehrungen/ST03_NOX_5pol_Zufuehrung, SFC *)
 PROGRAM ST03_NOX_5pol_Zufuehrung
VAR_OUTPUT
	SFCCurrentPOU			: STRING:='ST03_NOX_5pol_Zufuehrung';
	SFCCurrentStep			: STRING:='';
	FB_CurrentStepHistorie	: FB_CurrentStepHistorie;
	SFCTime					: DINT;
	State   				: StateObject	:= STATE_WAIT;
	Result  				: StateResult;
END_VAR
VAR_INPUT
	Start				:BOOL;
END_VAR
VAR
	MsgOK				: BOOL;
	MsgCancel			: BOOL;
	SFCRun				: BOOL;
	SFCTimeStart		: TIME;
	Delay				: TON;
	(* Userdefinded area *)

	i					: INT;
	RepeatCounter		: INT;
	NokCounter			: INT;
	NokCounterPercent	: INT;
  	NokPercent   		: ARRAY[1..100] OF BOOL;
END_VAR
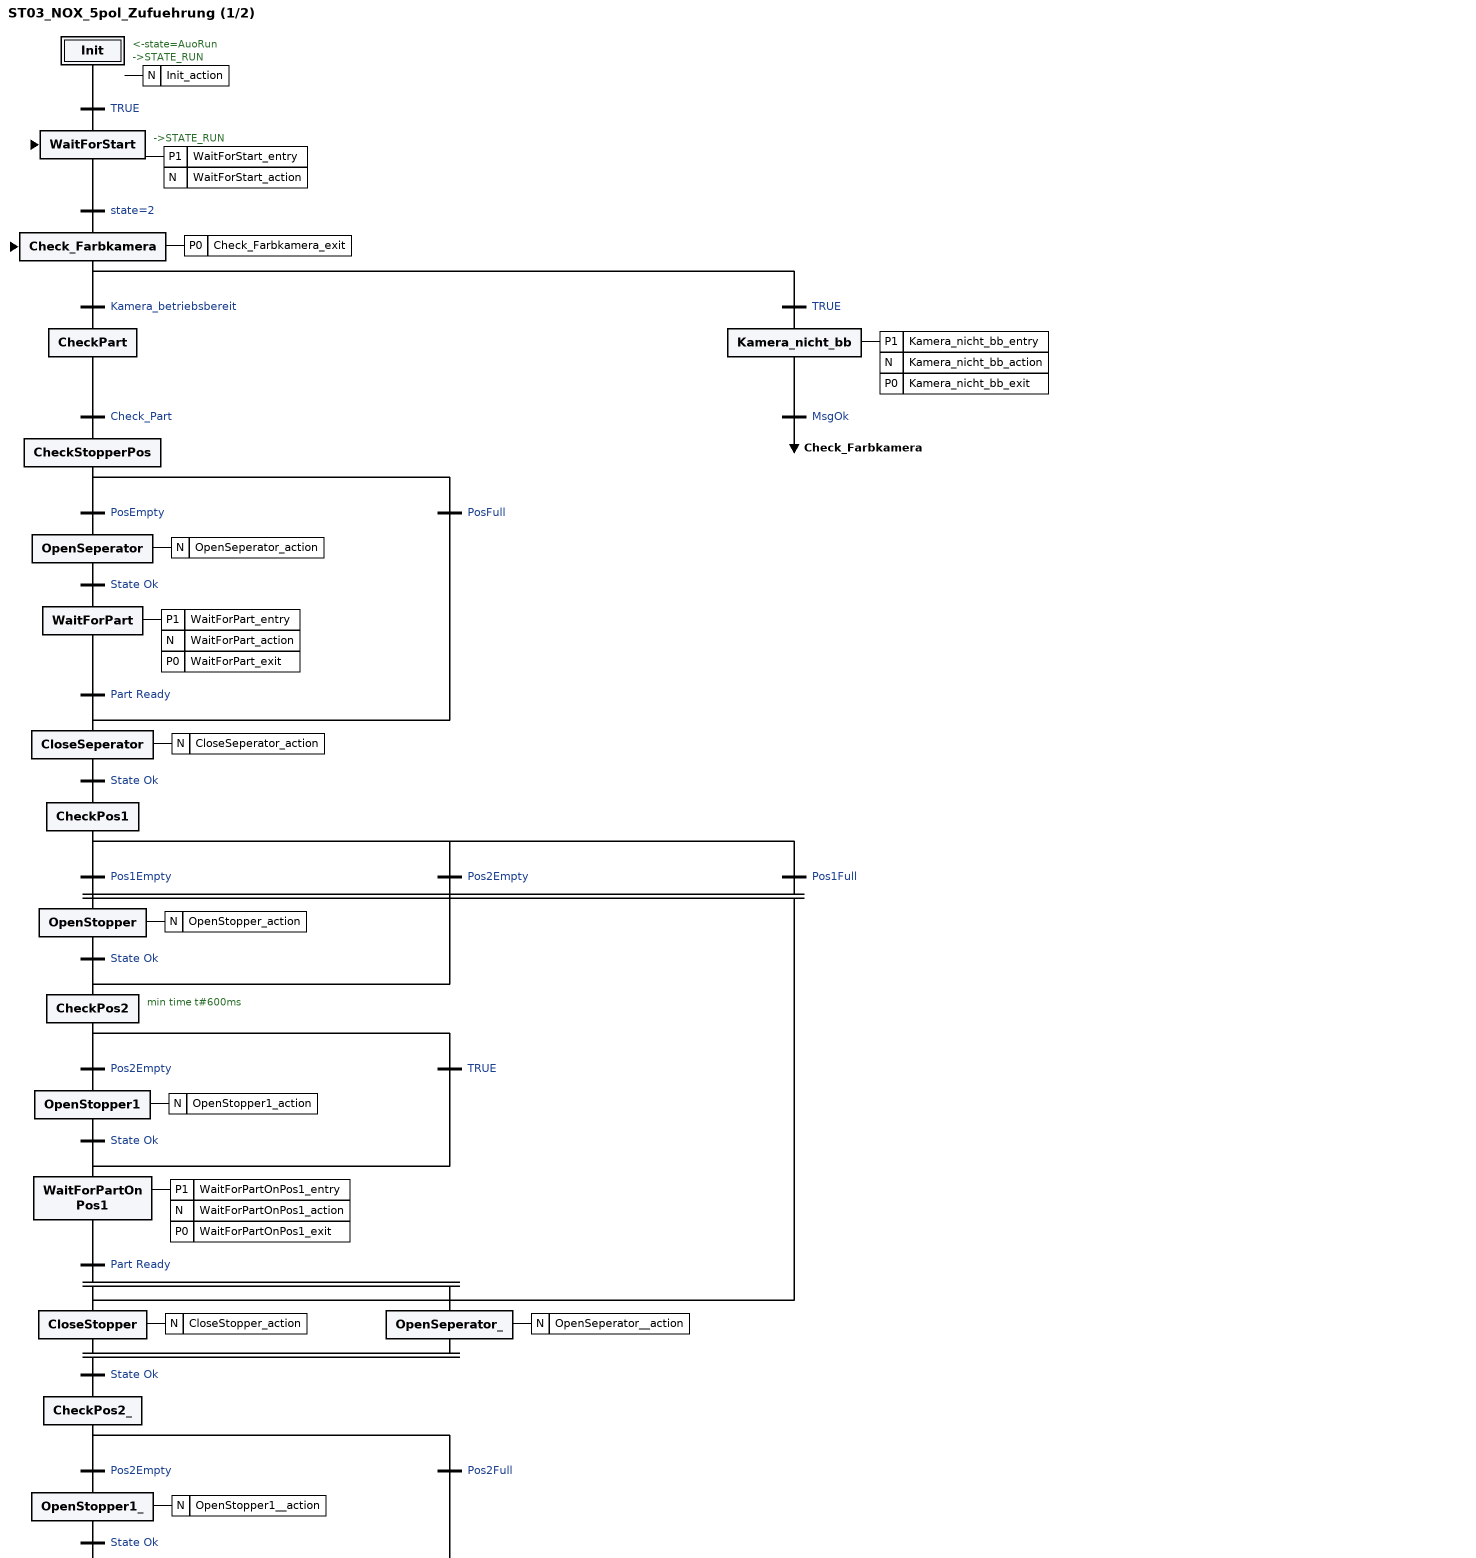
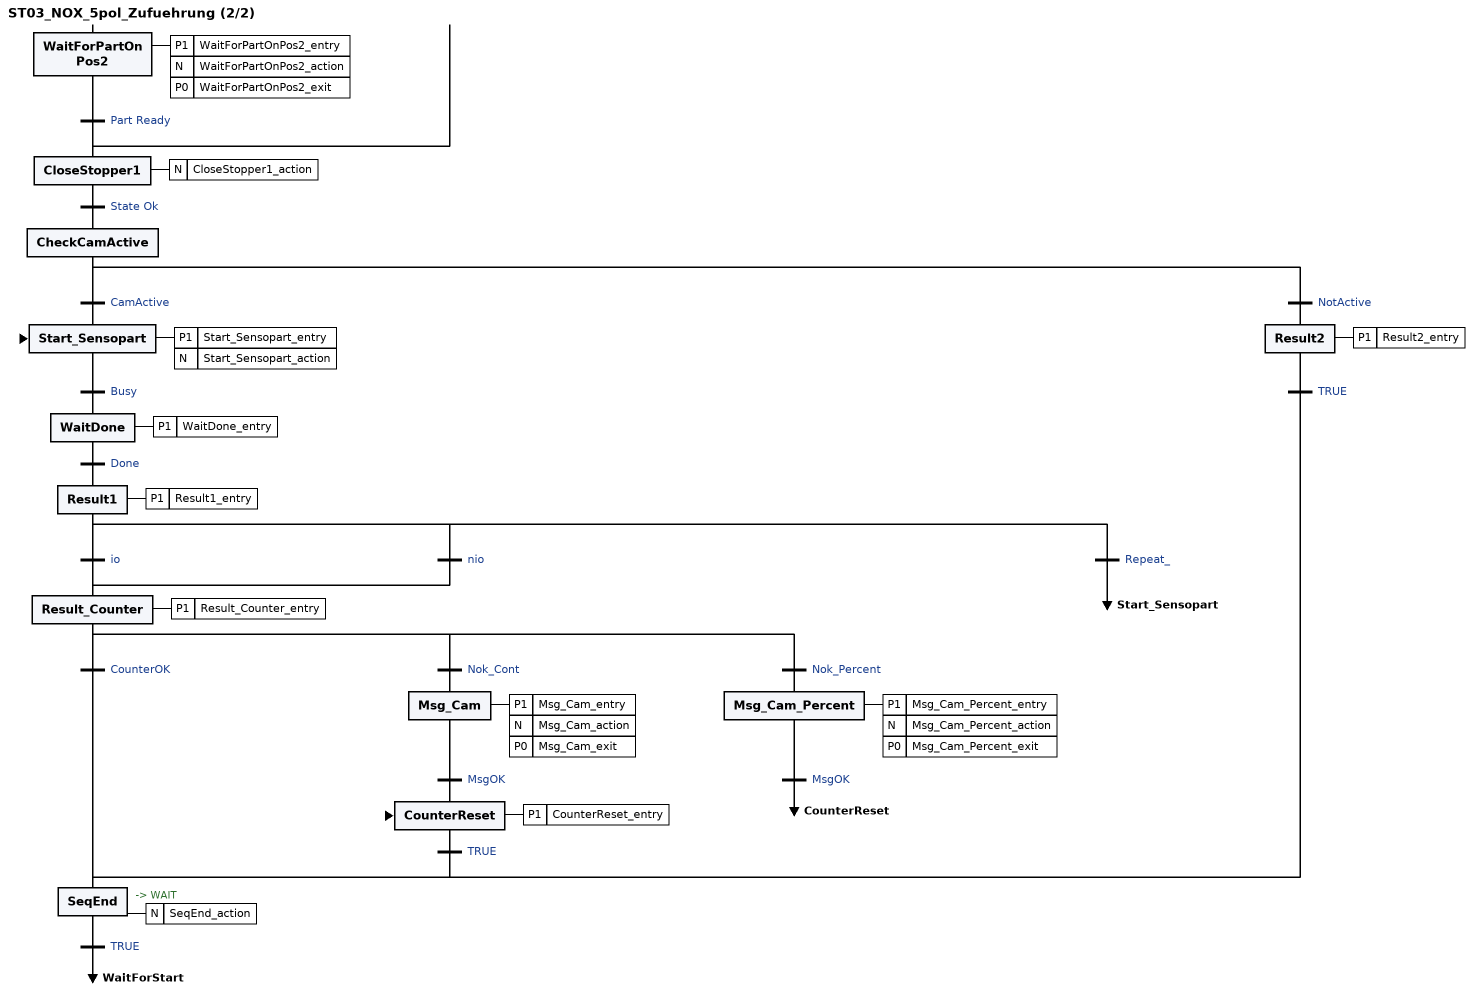
INITIAL_STEP Init: (* <-state=AuoRun / ->STATE_RUN *)
	Init_action(N);
END_STEP
TRANSITION FROM Init TO WaitForStart := TRUE;
END_TRANSITION
STEP WaitForStart: (* ->STATE_RUN *)
	WaitForStart_entry(P1);
	WaitForStart_action(N);
END_STEP
TRANSITION FROM WaitForStart TO Check_Farbkamera := state=2;
END_TRANSITION
STEP Check_Farbkamera:
	Check_Farbkamera_exit(P0);
END_STEP
TRANSITION FROM Check_Farbkamera TO CheckPart := Kamera_betriebsbereit;
END_TRANSITION
TRANSITION FROM Check_Farbkamera TO Kamera_nicht_bb := TRUE;
END_TRANSITION
STEP Kamera_nicht_bb:
	Kamera_nicht_bb_entry(P1);
	Kamera_nicht_bb_action(N);
	Kamera_nicht_bb_exit(P0);
END_STEP
TRANSITION FROM Kamera_nicht_bb TO Check_Farbkamera := MsgOk;
END_TRANSITION
STEP CheckPart:
END_STEP
TRANSITION FROM CheckPart TO CheckStopperPos := Check_Part;
END_TRANSITION
STEP CheckStopperPos:
END_STEP
TRANSITION FROM CheckStopperPos TO OpenSeperator := PosEmpty;
END_TRANSITION
TRANSITION FROM CheckStopperPos TO CloseSeperator := PosFull;
END_TRANSITION
STEP OpenSeperator:
	OpenSeperator_action(N);
END_STEP
TRANSITION FROM OpenSeperator TO WaitForPart := State Ok;
END_TRANSITION
STEP WaitForPart:
	WaitForPart_entry(P1);
	WaitForPart_action(N);
	WaitForPart_exit(P0);
END_STEP
TRANSITION FROM WaitForPart TO CloseSeperator := Part Ready;
END_TRANSITION
STEP CloseSeperator:
	CloseSeperator_action(N);
END_STEP
TRANSITION FROM CloseSeperator TO CheckPos1 := State Ok;
END_TRANSITION
STEP CheckPos1:
END_STEP
TRANSITION FROM CheckPos1 TO OpenStopper := Pos1Empty;
END_TRANSITION
TRANSITION FROM CheckPos1 TO CheckPos2 := Pos2Empty;
END_TRANSITION
TRANSITION FROM CheckPos1 TO (CloseStopper, OpenSeperator_) := Pos1Full;
END_TRANSITION
STEP OpenStopper:
	OpenStopper_action(N);
END_STEP
TRANSITION FROM OpenStopper TO CheckPos2 := State Ok;
END_TRANSITION
STEP CheckPos2: (* min time t#600ms *)
END_STEP
TRANSITION FROM CheckPos2 TO OpenStopper1 := Pos2Empty;
END_TRANSITION
TRANSITION FROM CheckPos2 TO WaitForPartOnPos1 := TRUE;
END_TRANSITION
STEP OpenStopper1:
	OpenStopper1_action(N);
END_STEP
TRANSITION FROM OpenStopper1 TO WaitForPartOnPos1 := State Ok;
END_TRANSITION
STEP WaitForPartOnPos1:
	WaitForPartOnPos1_entry(P1);
	WaitForPartOnPos1_action(N);
	WaitForPartOnPos1_exit(P0);
END_STEP
TRANSITION FROM WaitForPartOnPos1 TO (CloseStopper, OpenSeperator_) := Part Ready;
END_TRANSITION
STEP CloseStopper:
	CloseStopper_action(N);
END_STEP
STEP OpenSeperator_:
	OpenSeperator__action(N);
END_STEP
TRANSITION FROM (CloseStopper, OpenSeperator_) TO CheckPos2_ := State Ok;
END_TRANSITION
STEP CheckPos2_:
END_STEP
TRANSITION FROM CheckPos2_ TO OpenStopper1_ := Pos2Empty;
END_TRANSITION
TRANSITION FROM CheckPos2_ TO CloseStopper1 := Pos2Full;
END_TRANSITION
STEP OpenStopper1_:
	OpenStopper1__action(N);
END_STEP
TRANSITION FROM OpenStopper1_ TO WaitForPartOnPos2 := State Ok;
END_TRANSITION
STEP WaitForPartOnPos2:
	WaitForPartOnPos2_entry(P1);
	WaitForPartOnPos2_action(N);
	WaitForPartOnPos2_exit(P0);
END_STEP
TRANSITION FROM WaitForPartOnPos2 TO CloseStopper1 := Part Ready;
END_TRANSITION
STEP CloseStopper1:
	CloseStopper1_action(N);
END_STEP
TRANSITION FROM CloseStopper1 TO CheckCamActive := State Ok;
END_TRANSITION
STEP CheckCamActive:
END_STEP
TRANSITION FROM CheckCamActive TO Start_Sensopart := CamActive;
END_TRANSITION
TRANSITION FROM CheckCamActive TO Result2 := NotActive;
END_TRANSITION
STEP Start_Sensopart:
	Start_Sensopart_entry(P1);
	Start_Sensopart_action(N);
END_STEP
TRANSITION FROM Start_Sensopart TO WaitDone := Busy;
END_TRANSITION
STEP WaitDone:
	WaitDone_entry(P1);
END_STEP
TRANSITION FROM WaitDone TO Result1 := Done;
END_TRANSITION
STEP Result1:
	Result1_entry(P1);
END_STEP
TRANSITION FROM Result1 TO Result_Counter := io;
END_TRANSITION
TRANSITION FROM Result1 TO Result_Counter := nio;
END_TRANSITION
TRANSITION FROM Result1 TO Start_Sensopart := Repeat_;
END_TRANSITION
STEP Result_Counter:
	Result_Counter_entry(P1);
END_STEP
TRANSITION FROM Result_Counter TO SeqEnd := CounterOK;
END_TRANSITION
TRANSITION FROM Result_Counter TO Msg_Cam := Nok_Cont;
END_TRANSITION
TRANSITION FROM Result_Counter TO Msg_Cam_Percent := Nok_Percent;
END_TRANSITION
STEP Msg_Cam:
	Msg_Cam_entry(P1);
	Msg_Cam_action(N);
	Msg_Cam_exit(P0);
END_STEP
TRANSITION FROM Msg_Cam TO CounterReset := MsgOK;
END_TRANSITION
STEP CounterReset:
	CounterReset_entry(P1);
END_STEP
TRANSITION FROM CounterReset TO SeqEnd := TRUE;
END_TRANSITION
STEP Msg_Cam_Percent:
	Msg_Cam_Percent_entry(P1);
	Msg_Cam_Percent_action(N);
	Msg_Cam_Percent_exit(P0);
END_STEP
TRANSITION FROM Msg_Cam_Percent TO CounterReset := MsgOK;
END_TRANSITION
STEP Result2:
	Result2_entry(P1);
END_STEP
TRANSITION FROM Result2 TO SeqEnd := TRUE;
END_TRANSITION
STEP SeqEnd: (* -> WAIT *)
	SeqEnd_action(N);
END_STEP
TRANSITION FROM SeqEnd TO WaitForStart := TRUE;
END_TRANSITION

ACTION Init_action:
Start:=FALSE;
State:=STATE_WAIT;
MsgOK:=FALSE;
MsgCancel:=FALSE;
SFCRun:=FALSE;
Result:=RESULT_NON;
END_ACTION

ACTION WaitForStart_entry:
;
END_ACTION

ACTION WaitForStart_action:
IF 	Start   THEN
	State:=STATE_RUN;
	SFCTimeStart:=TIME();
	Start:=FALSE;
ELSE
	State:=STATE_WAIT;
	MsgOK:=FALSE;
	MsgCancel:=FALSE;
	SFCRun:=FALSE;
END_IF
END_ACTION

ACTION Check_Farbkamera_exit:
Result:=RESULT_NON;

IF NOT ST03_8_100_A1.Activated THEN
	Result:= RESULT_OK;
END_IF
END_ACTION

ACTION Kamera_nicht_bb_entry:
MessageHandler.ClearMessageLines(sVisu:=Visu.Message);
END_ACTION

ACTION Kamera_nicht_bb_action:
MessageHandler.Msg.ID:='PM152';
MessageHandler.Msg.Name:='Check Camera';
MessageHandler.Msg.Text:='Sesopart Kamera ist nicht betriebsbereit';
MessageHandler.Msg.Color:=Color.red;
MessageHandler.Msg.Station:=1;


MessageHandler(
	Prio:=2, 							(*1=highest, .. , 4=lowest*)
	Btn1Addr:=ADR(MsgOk),			(*Address of Button1 , if Zero then Button is unvisible*)
	Btn2Addr:=,						(*Address of Button2 , if Zero then Button is unvisible*)
	sVisu:=Visu.Message);
END_ACTION

ACTION Kamera_nicht_bb_exit:
MsgOk:=FALSE;
MsgCancel:=FALSE;
ST02_DT_95_A1.b_quitt:=TRUE;
END_ACTION

ACTION OpenSeperator_action:
ST03_4x3_Y70_5.MoveInit:=TRUE;		(*Zuführung Vereinzler AST/GST *)
END_ACTION

ACTION WaitForPart_entry:
ProcessMessage02:='';
Delay(IN:=FALSE);
END_ACTION

ACTION WaitForPart_action:
ProcessMessage02:='2IM6';				(*warte auf Teil Übergabeposition 1*)
Delay(	IN:=ST03_4x2_B69_5.BitInToCheck, (*ISK anwesend am Stopper*)
		PT:=T#50ms);
END_ACTION

ACTION WaitForPart_exit:
ProcessMessage02:='';
END_ACTION

ACTION CloseSeperator_action:
ST03_4x3_Y70_5.MoveWork:=TRUE;		(*Zuführung Vereinzler AST/GST *)
END_ACTION

ACTION OpenStopper_action:
ST03_4x3_Y70_6.MoveWork:=TRUE;		(*Zuführung Stopper AST/GST *)
END_ACTION

ACTION OpenStopper1_action:
ST03_4x3_Y70_7.MoveWork:=TRUE;		(* Zuführung Stopper Übergabeposition AST/GST*)
END_ACTION

ACTION WaitForPartOnPos1_entry:
ProcessMessage02:='';
Delay(IN:=FALSE);
END_ACTION

ACTION WaitForPartOnPos1_action:
ProcessMessage02:='2IM6';					(*warte auf Teil Übergabeposition 1*)
Delay.IN:=ST03_4x3_B70_0.BitInToCheck;  	(*ISK anwesend Übergabeposition Stopper *)

Delay.PT:=T#50ms;
Delay();
END_ACTION

ACTION WaitForPartOnPos1_exit:
ProcessMessage02:='';
END_ACTION

ACTION CloseStopper_action:
ST03_4x3_Y70_6.MoveInit:=TRUE;		(*Zuführung Stopper AST/GST *)
END_ACTION

ACTION OpenSeperator__action:
ST03_4x3_Y70_5.MoveInit:=TRUE;		(*Zuführung Vereinzler AST/GST *)
END_ACTION

ACTION OpenStopper1__action:
ST03_4x3_Y70_7.MoveWork:=TRUE;		(* Zuführung Stopper Übergabeposition AST/GST*)
END_ACTION

ACTION WaitForPartOnPos2_entry:
ProcessMessage02:='';
Delay(IN:=FALSE);
END_ACTION

ACTION WaitForPartOnPos2_action:
ProcessMessage02:='2IM5';						(*warte auf Teil Übergabeposition 2*)
Delay(	IN:=ST03_4x3_B70_1.BitInToCheck, 		(*ISK anwesend Übergabeposition *)
		PT:=T#50ms);
END_ACTION

ACTION WaitForPartOnPos2_exit:
ProcessMessage02:='';
END_ACTION

ACTION CloseStopper1_action:
ST03_4x3_Y70_7.MoveInit:=TRUE;		(* Zuführung Stopper Übergabeposition AST/GST *)
END_ACTION

ACTION Start_Sensopart_entry:
Result:=RESULT_NON;
END_ACTION

ACTION Start_Sensopart_action:
ST03_8_100_A1.JobNo := TD.Sensopart_CamProgNo ;
ST03_8_100_A1.st_ctrl_in.b_start := TRUE;
END_ACTION

ACTION WaitDone_entry:
ST03_8_100_A1.st_ctrl_in.b_start := FALSE;
RepeatCounter:=RepeatCounter+1;
END_ACTION

ACTION Result1_entry:
IF 	(ST03_8_100_A1.b_Kam_Pruef_IO AND	 (*Kamera Farberkennung*)
	NOT ST03_8_100_A1.b_Kam_Pruef_NIO)THEN
	Result:=RESULT_OK;
ELSE
	Result:=RESULT_NOK;
END_IF
END_ACTION

ACTION Result_Counter_entry:
IF 	(ST02_DT_95_A2.b_Kam_Pruef_IO AND	 (*Kamera Farberkennung*)
	NOT ST02_DT_95_A2.b_Kam_Pruef_NIO)THEN
	Result:=Result+10;
ELSE
	Result:=Result+90;
END_IF

FOR i:=100 TO 2 BY-1 DO
   NokPercent[i] := NokPercent[i-1];
END_FOR

IF	Result = 11 THEN
	NokCounter:=0;
	NokPercent[1] := FALSE;
	gRob01GripState:=PART_OK;
ELSE
	NokCounter:=NokCounter+1;
	NokPercent[1] := TRUE;
	gRob01GripState:=PART_NOK;
END_IF
END_ACTION

ACTION Msg_Cam_entry:
MessageHandler.ClearMessageLines(sVisu:=Visu.Message);
END_ACTION

ACTION Msg_Cam_action:
MessageHandler.Msg.ID:='PM112';
MessageHandler.Msg.Name:='Sensopart Kam.-Erg. Prüfung  n.i.o:';
MessageHandler.Msg.Text:='Sensopart Kam.-Erg. Prüfung  n.i.o: Fehler in Folge';
MessageHandler.Msg.Color:=Color.red;
MessageHandler.Msg.Station:=3;
MessageHandler.MsgButton1Text:='continue';

MessageHandler(
	Prio:=2, 								(*1=highest, .. , 4=lowest*)
	Btn1Addr:=ADR(MsgOk),				(*Address of Button1 , if Zero then Button is unvisible*)
	Btn2Addr:=0(*ADR(MsgCancel)*),			(*Address of Button2 , if Zero then Button is unvisible*)
	sVisu:=Visu.Message);
END_ACTION

ACTION Msg_Cam_exit:
MsgOk:=FALSE;
MsgCancel:=FALSE;
END_ACTION

ACTION CounterReset_entry:
NokCounter:=0;
(*Percent Register löschen*)
FOR i:=1 TO 100 BY 1 DO
  NokPercent[i]:= FALSE;
END_FOR
END_ACTION

ACTION Msg_Cam_Percent_entry:
MessageHandler.ClearMessageLines(sVisu:=Visu.Message);
END_ACTION

ACTION Msg_Cam_Percent_action:
MessageHandler.Msg.ID:='PM113';
MessageHandler.Msg.Name:='Sensopart Kam.-Erg. Prüfung  n.i.o:';
MessageHandler.Msg.Text:='Sensopart Kam.-Erg. Prüfung  n.i.o:% Fehler';
MessageHandler.Msg.Color:=Color.red;
MessageHandler.Msg.Station:=3;
MessageHandler.MsgButton1Text:='continue';

MessageHandler(
	Prio:=2, 								(*1=highest, .. , 4=lowest*)
	Btn1Addr:=ADR(MsgOk),				(*Address of Button1 , if Zero then Button is unvisible*)
	Btn2Addr:=0(*ADR(MsgCancel)*),			(*Address of Button2 , if Zero then Button is unvisible*)
	sVisu:=Visu.Message);
END_ACTION

ACTION Msg_Cam_Percent_exit:
MsgOk:=FALSE;
MsgCancel:=FALSE;
END_ACTION

ACTION Result2_entry:
Result:= RESULT_OK;
END_ACTION

ACTION SeqEnd_action:
SFCTime:=TIME_TO_DINT(TIME()-SFCTimeStart);
State:=STATE_WAIT;
END_ACTION

TRANSITION Kamera_betriebsbereit:
(*Kamera Farberkennung*)
(
NOT ST03_8_100_A1.sm_kamera_nicht_bb OR
NOT ST03_8_100_A1.Activated	)
END_TRANSITION

TRANSITION Check_Part:
Robot01.ActualArea <> 4 AND
(
NOT ST03_4x3_B70_0.BitInToCheck OR	(* ISK anwesend Übergabeposition Stopper*)
NOT ST03_4x3_B70_1.BitInToCheck )	(* ISK anwesend Übergabeposition*)
END_TRANSITION

TRANSITION PosEmpty:
NOT ST03_4x2_B69_5.BitInToCheck			 	(*  ISK anwesend am Stopper*)
END_TRANSITION

TRANSITION State Ok:
ST03_4x3_Y70_5.State=STATE_OK (*Zuführung Vereinzler AST/GST *)
END_TRANSITION

TRANSITION Part Ready:
Delay.Q
END_TRANSITION

TRANSITION PosFull:
ST03_4x2_B69_5.BitInToCheck			 	(*  ISK anwesend am Stopper*)
END_TRANSITION

TRANSITION State Ok:
ST03_4x3_Y70_5.State=STATE_OK (*Zuführung Vereinzler AST/GST *)
END_TRANSITION

TRANSITION Pos1Empty:
NOT ST03_4x3_B70_0.BitInToCheck AND 	(*  ISK anwesend Übergabeposition Stopper*)
ST03_4x2_B69_5.BitInToCheck			 	(*  ISK anwesend am Stopper*)
END_TRANSITION

TRANSITION Pos2Empty:
ST03_4x3_B70_0.BitInToCheck AND 	(*  ISK anwesend Übergabeposition Stopper*)
NOT ST03_4x3_B70_1.BitInToCheck AND 	(*  ISK anwesend Übergabeposition*)
ST03_4x2_B69_5.BitInToCheck			 	(*  ISK anwesend am Stopper*)
END_TRANSITION

TRANSITION State Ok:
ST03_4x3_Y70_6.State=STATE_OK 	(*Zuführung Stopper AST/GST *)
END_TRANSITION

TRANSITION Pos2Empty:
NOT ST03_4x3_B70_1.BitInToCheck AND 	(*  ISK anwesend Übergabeposition*)
NOT ST03_4x2_B69_5.BitInToCheck			 (*ISK anwesend am Stopper*)
END_TRANSITION

TRANSITION State Ok:
ST03_4x3_Y70_7.State=STATE_OK 	(* Zuführung Stopper Übergabeposition AST/GST *)
END_TRANSITION

TRANSITION Part Ready:
Delay.Q
END_TRANSITION

TRANSITION Pos1Full:
ST03_4x3_B70_0.BitInToCheck 	(*ISK anwesend Übergabeposition Stopper*)
END_TRANSITION

TRANSITION State Ok:
ST03_4x3_Y70_6.State=STATE_OK AND	(*Zuführung Stopper AST/GST *)
ST03_4x3_Y70_5.State=STATE_OK (*Zuführung Vereinzler AST/GST *)
END_TRANSITION

TRANSITION Pos2Empty:
NOT ST03_4x3_B70_1.BitInToCheck AND 	(*  ISK anwesend Übergabeposition*)
ST03_4x3_B70_0.BitInToCheck			 	(*  ISK anwesend Übergabeposition Stopper*)
END_TRANSITION

TRANSITION State Ok:
ST03_4x3_Y70_7.State=STATE_OK 	(* Zuführung Stopper Übergabeposition AST/GST *)
END_TRANSITION

TRANSITION Part Ready:
Delay.Q
END_TRANSITION

TRANSITION Pos2Full:
ST03_4x3_B70_1.BitInToCheck	 	(*ISK anwesend Übergabeposition*)
END_TRANSITION

TRANSITION State Ok:
ST03_4x3_Y70_7.State=STATE_OK 	(* Zuführung Stopper Übergabeposition AST/GST *)
END_TRANSITION

TRANSITION CamActive:
ST03_8_100_A1.Activated
END_TRANSITION

TRANSITION Busy:
ST03_8_100_A1.st_ctrl_out.b_busy (*Kamera Farberkennung Ehternet*)
END_TRANSITION

TRANSITION Done:
ST03_8_100_A1.st_ctrl_out.b_fertig
END_TRANSITION

TRANSITION io:
Result = RESULT_OK
END_TRANSITION

TRANSITION nio:
RepeatCounter>=2
END_TRANSITION

TRANSITION Repeat_:
TRUE
END_TRANSITION

TRANSITION CounterOK:
NokCounter<MP.ST03.CamNoOfErrors AND
NokCounterPercent < MP.ST02.CamNoOfErrorsPercent
END_TRANSITION

TRANSITION Nok_Cont:
NokCounter >= MP.ST03.CamNoOfErrors
END_TRANSITION

TRANSITION Nok_Percent:
NokCounterPercent >= MP.ST03.CamNoOfErrorsPercent
END_TRANSITION

TRANSITION NotActive:
TRUE
END_TRANSITION
END_PROGRAM

(* POU Stations/ST_03_Ruestsaetze/ST_03_SFCs/Zufuehrungen/ST03_NOX_6pol_Zufuehrung, SFC *)
 PROGRAM ST03_NOX_6pol_Zufuehrung

VAR_OUTPUT
	SFCCurrentPOU			: STRING:='ST03_NOX_6pol_Zufuehrung';
	SFCCurrentStep			: STRING:='';
	FB_CurrentStepHistorie	: FB_CurrentStepHistorie;
	SFCTime					: DINT;
	State   				: StateObject	:= STATE_WAIT;
	Result  				: StateResult;
	LockForCam				: BOOL;

END_VAR
VAR_INPUT
	Start					: BOOL;
END_VAR
VAR
	MsgOK					: BOOL;
	MsgCancel				: BOOL;
	SFCRun					: BOOL;
	SFCTimeStart			: TIME;
	Delay					: TON;
	(* Userdefinded area *)

	i						: INT;
	RepeatCounter			: INT;
	NokCounter_Cam			: ARRAY[1..2] OF INT;
	NokCounterPercent_Cam	: ARRAY[1..2] OF INT;
  	NokPercent_Cam  		: ARRAY[1..2, 1..100] OF BOOL;

	Result_Cam1				: ARRAY[1..2] OF StateResult;
	Result_Cam2				: StateResult;
	Part					: INT := 0;	(*Teil 1 oder Teil 2*)

	KeyenceCam_AlwaysOK		: BOOL:=FALSE; (*Keyence RESULT_OK - nur für IBN*)
	SensopartCam_AlwaysOK	: BOOL:=FALSE; (*Sensopart RESULT_OK - nur für IBN*)
END_VAR
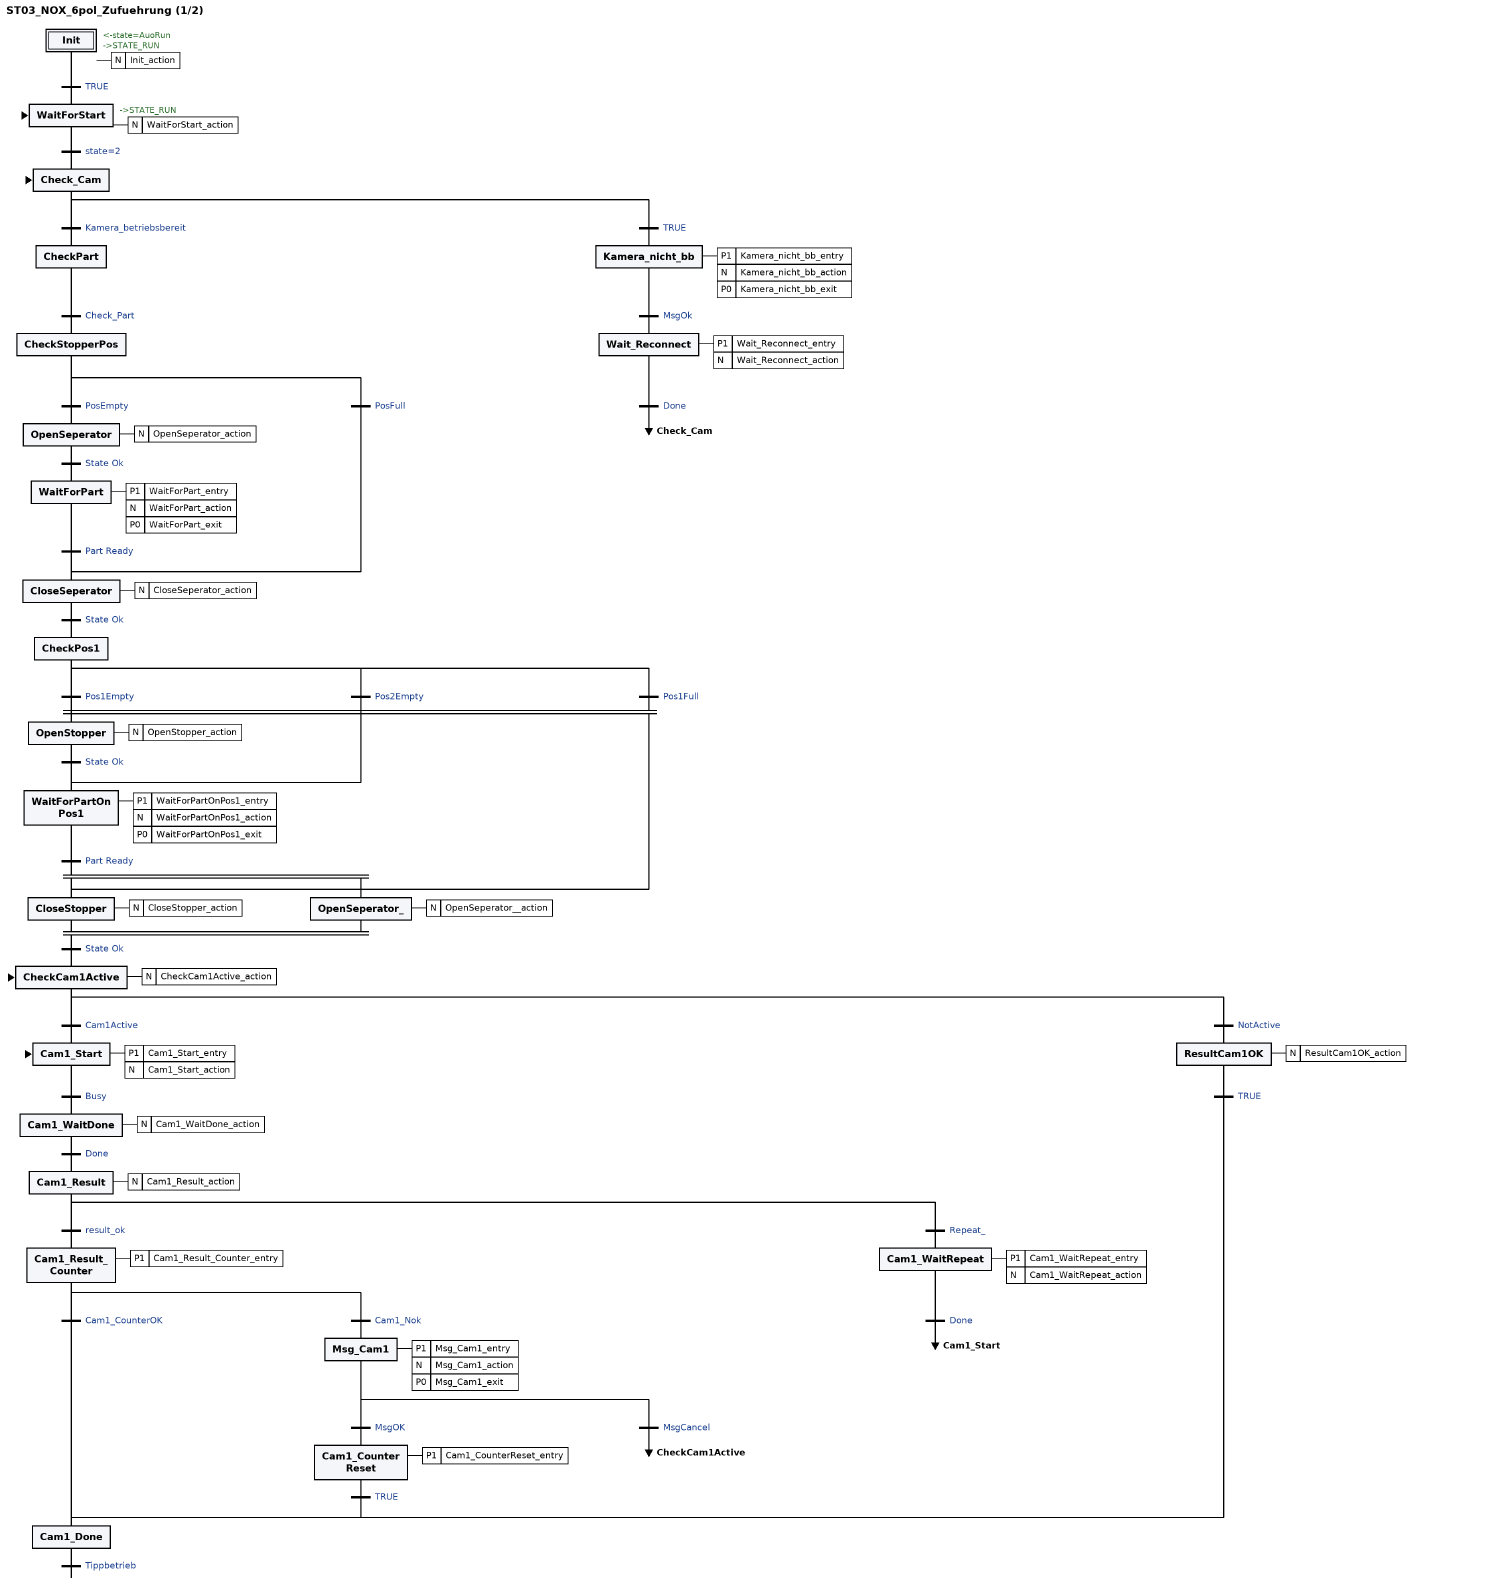
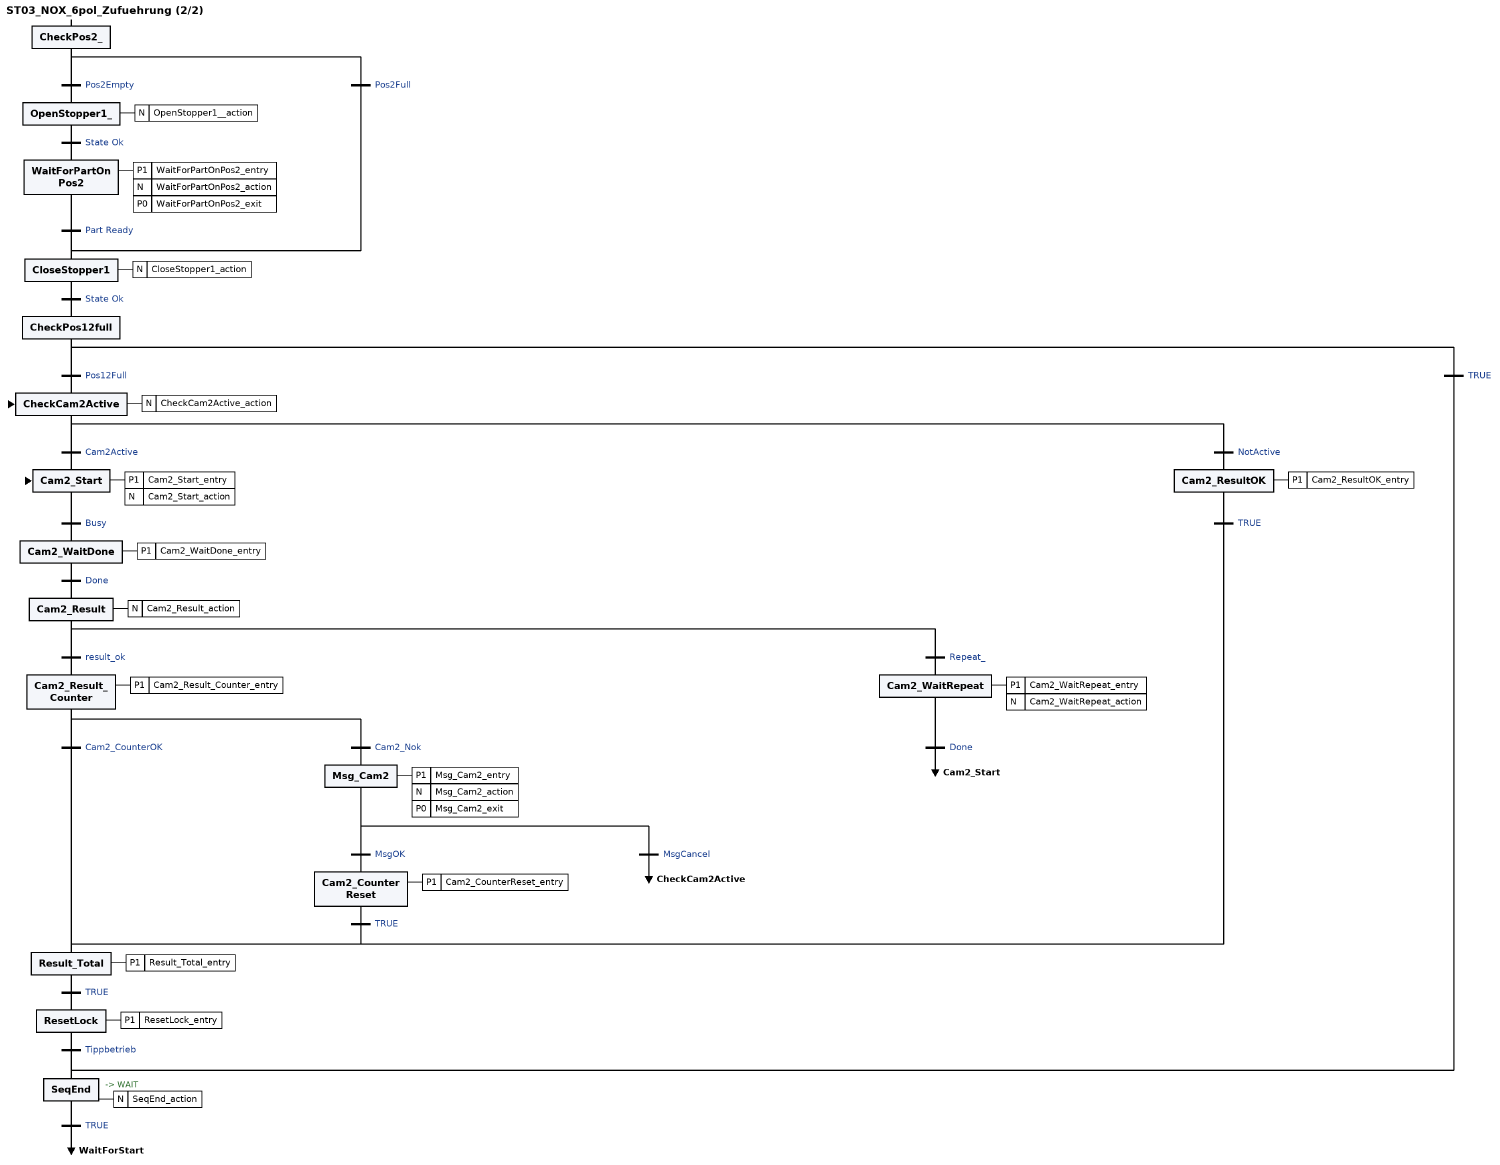
INITIAL_STEP Init: (* <-state=AuoRun / ->STATE_RUN *)
	Init_action(N);
END_STEP
TRANSITION FROM Init TO WaitForStart := TRUE;
END_TRANSITION
STEP WaitForStart: (* ->STATE_RUN *)
	WaitForStart_action(N);
END_STEP
TRANSITION FROM WaitForStart TO Check_Cam := state=2;
END_TRANSITION
STEP Check_Cam:
END_STEP
TRANSITION FROM Check_Cam TO CheckPart := Kamera_betriebsbereit;
END_TRANSITION
TRANSITION FROM Check_Cam TO Kamera_nicht_bb := TRUE;
END_TRANSITION
STEP Kamera_nicht_bb:
	Kamera_nicht_bb_entry(P1);
	Kamera_nicht_bb_action(N);
	Kamera_nicht_bb_exit(P0);
END_STEP
TRANSITION FROM Kamera_nicht_bb TO Wait_Reconnect := MsgOk;
END_TRANSITION
STEP Wait_Reconnect:
	Wait_Reconnect_entry(P1);
	Wait_Reconnect_action(N);
END_STEP
TRANSITION FROM Wait_Reconnect TO Check_Cam := Done;
END_TRANSITION
STEP CheckPart:
END_STEP
TRANSITION FROM CheckPart TO CheckStopperPos := Check_Part;
END_TRANSITION
STEP CheckStopperPos:
END_STEP
TRANSITION FROM CheckStopperPos TO OpenSeperator := PosEmpty;
END_TRANSITION
TRANSITION FROM CheckStopperPos TO CloseSeperator := PosFull;
END_TRANSITION
STEP OpenSeperator:
	OpenSeperator_action(N);
END_STEP
TRANSITION FROM OpenSeperator TO WaitForPart := State Ok;
END_TRANSITION
STEP WaitForPart:
	WaitForPart_entry(P1);
	WaitForPart_action(N);
	WaitForPart_exit(P0);
END_STEP
TRANSITION FROM WaitForPart TO CloseSeperator := Part Ready;
END_TRANSITION
STEP CloseSeperator:
	CloseSeperator_action(N);
END_STEP
TRANSITION FROM CloseSeperator TO CheckPos1 := State Ok;
END_TRANSITION
STEP CheckPos1:
END_STEP
TRANSITION FROM CheckPos1 TO OpenStopper := Pos1Empty;
END_TRANSITION
TRANSITION FROM CheckPos1 TO WaitForPartOnPos1 := Pos2Empty;
END_TRANSITION
TRANSITION FROM CheckPos1 TO (CloseStopper, OpenSeperator_) := Pos1Full;
END_TRANSITION
STEP OpenStopper:
	OpenStopper_action(N);
END_STEP
TRANSITION FROM OpenStopper TO WaitForPartOnPos1 := State Ok;
END_TRANSITION
STEP WaitForPartOnPos1:
	WaitForPartOnPos1_entry(P1);
	WaitForPartOnPos1_action(N);
	WaitForPartOnPos1_exit(P0);
END_STEP
TRANSITION FROM WaitForPartOnPos1 TO (CloseStopper, OpenSeperator_) := Part Ready;
END_TRANSITION
STEP CloseStopper:
	CloseStopper_action(N);
END_STEP
STEP OpenSeperator_:
	OpenSeperator__action(N);
END_STEP
TRANSITION FROM (CloseStopper, OpenSeperator_) TO CheckCam1Active := State Ok;
END_TRANSITION
STEP CheckCam1Active:
	CheckCam1Active_action(N);
END_STEP
TRANSITION FROM CheckCam1Active TO Cam1_Start := Cam1Active;
END_TRANSITION
TRANSITION FROM CheckCam1Active TO ResultCam1OK := NotActive;
END_TRANSITION
STEP Cam1_Start:
	Cam1_Start_entry(P1);
	Cam1_Start_action(N);
END_STEP
TRANSITION FROM Cam1_Start TO Cam1_WaitDone := Busy;
END_TRANSITION
STEP Cam1_WaitDone:
	Cam1_WaitDone_action(N);
END_STEP
TRANSITION FROM Cam1_WaitDone TO Cam1_Result := Done;
END_TRANSITION
STEP Cam1_Result:
	Cam1_Result_action(N);
END_STEP
TRANSITION FROM Cam1_Result TO Cam1_Result_Counter := result_ok;
END_TRANSITION
TRANSITION FROM Cam1_Result TO Cam1_WaitRepeat := Repeat_;
END_TRANSITION
STEP Cam1_WaitRepeat:
	Cam1_WaitRepeat_entry(P1);
	Cam1_WaitRepeat_action(N);
END_STEP
TRANSITION FROM Cam1_WaitRepeat TO Cam1_Start := Done;
END_TRANSITION
STEP Cam1_Result_Counter:
	Cam1_Result_Counter_entry(P1);
END_STEP
TRANSITION FROM Cam1_Result_Counter TO Cam1_Done := Cam1_CounterOK;
END_TRANSITION
TRANSITION FROM Cam1_Result_Counter TO Msg_Cam1 := Cam1_Nok;
END_TRANSITION
STEP Msg_Cam1:
	Msg_Cam1_entry(P1);
	Msg_Cam1_action(N);
	Msg_Cam1_exit(P0);
END_STEP
TRANSITION FROM Msg_Cam1 TO Cam1_CounterReset := MsgOK;
END_TRANSITION
TRANSITION FROM Msg_Cam1 TO CheckCam1Active := MsgCancel;
END_TRANSITION
STEP Cam1_CounterReset:
	Cam1_CounterReset_entry(P1);
END_STEP
TRANSITION FROM Cam1_CounterReset TO Cam1_Done := TRUE;
END_TRANSITION
STEP ResultCam1OK:
	ResultCam1OK_action(N);
END_STEP
TRANSITION FROM ResultCam1OK TO Cam1_Done := TRUE;
END_TRANSITION
STEP Cam1_Done:
END_STEP
TRANSITION FROM Cam1_Done TO CheckPos2_ := Tippbetrieb;
END_TRANSITION
STEP CheckPos2_:
END_STEP
TRANSITION FROM CheckPos2_ TO OpenStopper1_ := Pos2Empty;
END_TRANSITION
TRANSITION FROM CheckPos2_ TO CloseStopper1 := Pos2Full;
END_TRANSITION
STEP OpenStopper1_:
	OpenStopper1__action(N);
END_STEP
TRANSITION FROM OpenStopper1_ TO WaitForPartOnPos2 := State Ok;
END_TRANSITION
STEP WaitForPartOnPos2:
	WaitForPartOnPos2_entry(P1);
	WaitForPartOnPos2_action(N);
	WaitForPartOnPos2_exit(P0);
END_STEP
TRANSITION FROM WaitForPartOnPos2 TO CloseStopper1 := Part Ready;
END_TRANSITION
STEP CloseStopper1:
	CloseStopper1_action(N);
END_STEP
TRANSITION FROM CloseStopper1 TO CheckPos12full := State Ok;
END_TRANSITION
STEP CheckPos12full:
END_STEP
TRANSITION FROM CheckPos12full TO CheckCam2Active := Pos12Full;
END_TRANSITION
TRANSITION FROM CheckPos12full TO SeqEnd := TRUE;
END_TRANSITION
STEP CheckCam2Active:
	CheckCam2Active_action(N);
END_STEP
TRANSITION FROM CheckCam2Active TO Cam2_Start := Cam2Active;
END_TRANSITION
TRANSITION FROM CheckCam2Active TO Cam2_ResultOK := NotActive;
END_TRANSITION
STEP Cam2_Start:
	Cam2_Start_entry(P1);
	Cam2_Start_action(N);
END_STEP
TRANSITION FROM Cam2_Start TO Cam2_WaitDone := Busy;
END_TRANSITION
STEP Cam2_WaitDone:
	Cam2_WaitDone_entry(P1);
END_STEP
TRANSITION FROM Cam2_WaitDone TO Cam2_Result := Done;
END_TRANSITION
STEP Cam2_Result:
	Cam2_Result_action(N);
END_STEP
TRANSITION FROM Cam2_Result TO Cam2_Result_Counter := result_ok;
END_TRANSITION
TRANSITION FROM Cam2_Result TO Cam2_WaitRepeat := Repeat_;
END_TRANSITION
STEP Cam2_Result_Counter:
	Cam2_Result_Counter_entry(P1);
END_STEP
TRANSITION FROM Cam2_Result_Counter TO Result_Total := Cam2_CounterOK;
END_TRANSITION
TRANSITION FROM Cam2_Result_Counter TO Msg_Cam2 := Cam2_Nok;
END_TRANSITION
STEP Msg_Cam2:
	Msg_Cam2_entry(P1);
	Msg_Cam2_action(N);
	Msg_Cam2_exit(P0);
END_STEP
TRANSITION FROM Msg_Cam2 TO Cam2_CounterReset := MsgOK;
END_TRANSITION
TRANSITION FROM Msg_Cam2 TO CheckCam2Active := MsgCancel;
END_TRANSITION
STEP Cam2_CounterReset:
	Cam2_CounterReset_entry(P1);
END_STEP
TRANSITION FROM Cam2_CounterReset TO Result_Total := TRUE;
END_TRANSITION
STEP Cam2_WaitRepeat:
	Cam2_WaitRepeat_entry(P1);
	Cam2_WaitRepeat_action(N);
END_STEP
TRANSITION FROM Cam2_WaitRepeat TO Cam2_Start := Done;
END_TRANSITION
STEP Cam2_ResultOK:
	Cam2_ResultOK_entry(P1);
END_STEP
TRANSITION FROM Cam2_ResultOK TO Result_Total := TRUE;
END_TRANSITION
STEP Result_Total:
	Result_Total_entry(P1);
END_STEP
TRANSITION FROM Result_Total TO ResetLock := TRUE;
END_TRANSITION
STEP ResetLock:
	ResetLock_entry(P1);
END_STEP
TRANSITION FROM ResetLock TO SeqEnd := Tippbetrieb;
END_TRANSITION
STEP SeqEnd: (* -> WAIT *)
	SeqEnd_action(N);
END_STEP
TRANSITION FROM SeqEnd TO WaitForStart := TRUE;
END_TRANSITION

ACTION Init_action:
Start:=FALSE;
State:=STATE_WAIT;
MsgOK:=FALSE;
MsgCancel:=FALSE;
SFCRun:=FALSE;
Result:=RESULT_NON;
LockForCam:=FALSE;
END_ACTION

ACTION WaitForStart_action:
IF 	Start   THEN
	State:=STATE_RUN;
	SFCTimeStart:=TIME();
	Start:=FALSE;
ELSE
	State:=STATE_WAIT;
	MsgOK:=FALSE;
	MsgCancel:=FALSE;
	SFCRun:=FALSE;
END_IF
END_ACTION

ACTION Kamera_nicht_bb_entry:
MessageHandler.ClearMessageLines(sVisu:=Visu.Message);
END_ACTION

ACTION Kamera_nicht_bb_action:
(* Sensopart Kamera *)
IF	ST03_8_100_A1.Activated AND
	ST03_8_100_A1.sm_kamera_nicht_bb THEN
	MessageHandler.Msg.ID:='PM152';
	MessageHandler.Msg.Text:='Sesopart Kamera ist nicht betriebsbereit';

(* Keyence Kamera *)
ELSIF
	ST03_8_105_A1.sConfig.Aktiv AND
	ST03_8_105_A1.sm_kamera_nicht_bb THEN
	MessageHandler.Msg.ID:='PM159';
	MessageHandler.Msg.Text:='Keyence Kamera ist nicht betriebsbereit';
END_IF

	MessageHandler.Msg.Name:='Check Camera';
	MessageHandler.Msg.Color:=Color.red;
	MessageHandler.Msg.Station:=1;

	MessageHandler(
		Prio:=2, 							(*1=highest, .. , 4=lowest*)
		Btn1Addr:=ADR(MsgOk),			(*Address of Button1 , if Zero then Button is unvisible*)
		Btn2Addr:=,						(*Address of Button2 , if Zero then Button is unvisible*)
		sVisu:=Visu.Message);
END_ACTION

ACTION Kamera_nicht_bb_exit:
MsgOk:=FALSE;
MsgCancel:=FALSE;

(* Sensopart Kamera *)
IF ST03_8_100_A1.Activated THEN
	ST03_8_100_A1.st_ctrl_in.b_quitt := TRUE;
END_IF

(* Keyence Kamera *)
IF ST03_8_105_A1.sConfig.Aktiv THEN
	ST03_8_105_A1.st_ctrl_in.b_quitt := TRUE;
END_IF
END_ACTION

ACTION Wait_Reconnect_entry:
Delay(IN:=FALSE);
END_ACTION

ACTION Wait_Reconnect_action:
Delay(	IN:=TRUE, 		(*warte kurz, um neu zu verbinden *)
		PT:=T#1s);
END_ACTION

ACTION OpenSeperator_action:
ST03_4x3_Y70_5.MoveInit:=TRUE;		(*Zuführung Vereinzler AST/GST *)
END_ACTION

ACTION WaitForPart_entry:
ProcessMessage02:='';
Delay(IN:=FALSE);
END_ACTION

ACTION WaitForPart_action:
ProcessMessage02:='2IM6';				(*warte auf Teil Übergabeposition 1*)
Delay(	IN:=ST03_4x2_B69_5.BitInToCheck, (*ISK anwesend am Stopper*)
		PT:=T#50ms);
END_ACTION

ACTION WaitForPart_exit:
ProcessMessage02:='';
END_ACTION

ACTION CloseSeperator_action:
ST03_4x3_Y70_5.MoveWork:=TRUE;		(*Zuführung Vereinzler AST/GST *)
END_ACTION

ACTION OpenStopper_action:
ST03_4x3_Y70_6.MoveWork:=TRUE;		(*Zuführung Stopper AST/GST *)
END_ACTION

ACTION WaitForPartOnPos1_entry:
ProcessMessage02:='';
Delay(IN:=FALSE);
END_ACTION

ACTION WaitForPartOnPos1_action:
ProcessMessage02:='2IM6';					(*warte auf Teil Übergabeposition 1*)
Delay.IN:=ST03_4x3_B70_0.BitInToCheck;  	(*ISK anwesend Übergabeposition Stopper *)

Delay.PT:=T#50ms;
Delay();
END_ACTION

ACTION WaitForPartOnPos1_exit:
ProcessMessage02:='';
END_ACTION

ACTION CloseStopper_action:
ST03_4x3_Y70_6.MoveInit:=TRUE;		(*Zuführung Stopper AST/GST *)
END_ACTION

ACTION OpenSeperator__action:
ST03_4x3_Y70_5.MoveInit:=TRUE;		(*Zuführung Vereinzler AST/GST *)
END_ACTION

ACTION CheckCam1Active_action:
RepeatCounter:=0;

(* Teil 1 oder Teil 2*)
IF 	NOT ST03_4x3_B70_1.BitInToCheck AND		(* Teil vor Stopper bzw. Übergabeposition 1*)
	ST03_4x3_B70_0.BitInToCheck THEN		(* Teil nach Stopper bzw. Übergabeposition 2*)
	Part := 1;
ELSE
	Part := 2;
END_IF

LockForCam:=TRUE;
END_ACTION

ACTION Cam1_Start_entry:
Result_Cam1[Part] := RESULT_NON;
END_ACTION

ACTION Cam1_Start_action:
ST03_8_105_A1.JobNo := TD.Keyence_CamProgNo ;		(* Keyence Kameraprogramm*)
ST03_8_105_A1.st_ctrl_in.b_start := TRUE;
END_ACTION

ACTION Cam1_WaitDone_action:
ST03_8_105_A1.st_ctrl_in.b_start := FALSE;
RepeatCounter:=RepeatCounter+1;
END_ACTION

ACTION Cam1_Result_action:
IF 	(ST03_8_105_A1.b_Kam_Pruef_IO AND			 (*Kamera 1 = Keyence IV4*)
	NOT ST03_8_105_A1.b_Kam_Pruef_NIO) OR
	KeyenceCam_AlwaysOK THEN
	Result_Cam1[Part] := RESULT_OK;
ELSE
	Result_Cam1[Part] := RESULT_NOK;
END_IF
END_ACTION

ACTION Cam1_WaitRepeat_entry:
Delay(IN:=FALSE);
END_ACTION

ACTION Cam1_WaitRepeat_action:
Delay(	IN:=TRUE, 		(*warte kurz, bevor neues Bild gemacht wird *)
		PT:=T#500ms);
END_ACTION

ACTION Cam1_Result_Counter_entry:
FOR i:=100 TO 2 BY-1 DO
   NokPercent_Cam[1,i] := NokPercent_Cam[1,i-1];
END_FOR

IF 	Result_Cam1[Part] = RESULT_NOK THEN
	NokCounter_Cam[1] := NokCounter_Cam[1] + 1;
	NokPercent_Cam[1,1] := TRUE;
ELSE
	NokCounter_Cam[1] := 0;
	NokPercent_Cam[1,1] := FALSE;
END_IF

(*Anzahl der Schlechtteile von den letzten 100 Prüfungen*)
NokCounterPercent_Cam[1] := 0;
FOR i:=1 TO 100 BY 1 DO
	IF NokPercent_Cam[1,i] THEN
	NokCounterPercent_Cam[1] := NokCounterPercent_Cam[1]+1;
	END_IF
END_FOR
END_ACTION

ACTION Msg_Cam1_entry:
MessageHandler.ClearMessageLines(sVisu:=Visu.Message);
END_ACTION

ACTION Msg_Cam1_action:
IF NokCounter_Cam[1] >= MP.ST03.CamNoOfErrors_KYE THEN
	MessageHandler.Msg.ID:='PM124';
	MessageHandler.Msg.Name:='Keyence Kam.-Erg. Prüfung  n.i.o:';
	MessageHandler.Msg.Text:='Keyence Kam.-Erg. Prüfung  n.i.o: Fehler in Folge';

ELSIF NokCounterPercent_Cam[1] >= MP.ST03.CamNoOfErrorsPercent_KYE THEN
	MessageHandler.Msg.ID:='PM125';
	MessageHandler.Msg.Name:='Keyence Kam.-Erg. Prüfung  n.i.o:';
	MessageHandler.Msg.Text:='Keyence Kam.-Erg. Prüfung  n.i.o:% Fehler';

END_IF

	MessageHandler.Msg.Color:=Color.red;
	MessageHandler.Msg.Station:=3;
	MessageHandler.MsgButton1Text:='continue';
	MessageHandler.MsgButton2Text:='repeat';
	
	MessageHandler(
		Prio:=2, 								(*1=highest, .. , 4=lowest*)
		Btn1Addr:=ADR(MsgOk),				(*Address of Button1 , if Zero then Button is unvisible*)
		Btn2Addr:=ADR(MsgCancel),			(*Address of Button2 , if Zero then Button is unvisible*)
		sVisu:=Visu.Message);
END_ACTION

ACTION Msg_Cam1_exit:
MsgOk:=FALSE;
MsgCancel:=FALSE;
END_ACTION

ACTION Cam1_CounterReset_entry:
NokCounter_Cam[1] := 0;
NokCounterPercent_Cam[1] := 0;
(*Percent Register löschen*)
FOR i:=1 TO 100 BY 1 DO
  NokPercent_Cam[1,i]:= FALSE;
END_FOR
END_ACTION

ACTION ResultCam1OK_action:
Result_Cam1[1] := RESULT_OK;
Result_Cam1[2] := RESULT_OK;
END_ACTION

ACTION OpenStopper1__action:
ST03_4x3_Y70_7.MoveWork:=TRUE;		(* Zuführung Stopper Übergabeposition AST/GST*)
END_ACTION

ACTION WaitForPartOnPos2_entry:
ProcessMessage02:='';
Delay(IN:=FALSE);
END_ACTION

ACTION WaitForPartOnPos2_action:
ProcessMessage02:='2IM5';						(*warte auf Teil Übergabeposition 2*)
Delay(	IN:=ST03_4x3_B70_1.BitInToCheck, 		(*ISK anwesend Übergabeposition *)
		PT:=T#50ms);
END_ACTION

ACTION WaitForPartOnPos2_exit:
ProcessMessage02:='';
END_ACTION

ACTION CloseStopper1_action:
ST03_4x3_Y70_7.MoveInit:=TRUE;		(* Zuführung Stopper Übergabeposition AST/GST *)
END_ACTION

ACTION CheckCam2Active_action:
RepeatCounter:=0;
END_ACTION

ACTION Cam2_Start_entry:
Result_Cam2 := RESULT_NON;
END_ACTION

ACTION Cam2_Start_action:
ST03_8_100_A1.JobNo := TD.Sensopart_CamProgNo ;
ST03_8_100_A1.st_ctrl_in.b_start := TRUE;
END_ACTION

ACTION Cam2_WaitDone_entry:
ST03_8_100_A1.st_ctrl_in.b_start := FALSE;
RepeatCounter:=RepeatCounter+1;
END_ACTION

ACTION Cam2_Result_action:
IF 	(ST03_8_100_A1.b_Kam_Pruef_IO AND			 (*Kamera 2 = Sensopart V20*)
	NOT ST03_8_100_A1.b_Kam_Pruef_NIO) OR
	SensopartCam_AlwaysOK THEN
	Result_Cam2 := RESULT_OK;
ELSE
	Result_Cam2 := RESULT_NOK;
END_IF
END_ACTION

ACTION Cam2_Result_Counter_entry:
FOR i:=100 TO 2 BY-1 DO
   NokPercent_Cam[2,i] := NokPercent_Cam[2,i-1];
END_FOR

IF	Result_Cam2 = RESULT_OK THEN
	NokCounter_Cam[2] := 0;
	NokPercent_Cam[2,1] := FALSE;
ELSE
	NokCounter_Cam[2] := NokCounter_Cam[2] + 1;
	NokPercent_Cam[2,1] := TRUE;
END_IF

(*Anzahl der Schlechtteile von den letzten 100 Prüfungen*)
NokCounterPercent_Cam[2] := 0;
FOR i:=1 TO 100 BY 1 DO
	IF NokPercent_Cam[2,i] THEN
	NokCounterPercent_Cam[2] := NokCounterPercent_Cam[2]+1;
	END_IF
END_FOR
END_ACTION

ACTION Msg_Cam2_entry:
MessageHandler.ClearMessageLines(sVisu:=Visu.Message);
END_ACTION

ACTION Msg_Cam2_action:
IF NokCounter_Cam[2] >= MP.ST03.CamNoOfErrors THEN
	MessageHandler.Msg.ID:='PM112';
	MessageHandler.Msg.Name:='Sensopart Kam.-Erg. Prüfung  n.i.o:';
	MessageHandler.Msg.Text:='Sensopart Kam.-Erg. Prüfung  n.i.o: Fehler in Folge';

ELSIF NokCounterPercent_Cam[2] >= MP.ST03.CamNoOfErrorsPercent THEN
	MessageHandler.Msg.ID:='PM113';
	MessageHandler.Msg.Name:='Sensopart Kam.-Erg. Prüfung  n.i.o:';
	MessageHandler.Msg.Text:='Sensopart Kam.-Erg. Prüfung  n.i.o:% Fehler';
END_IF

	MessageHandler.Msg.Color:=Color.red;
	MessageHandler.Msg.Station:=3;
	MessageHandler.MsgButton1Text:='continue';
	MessageHandler.MsgButton2Text:='repeat';
	
	MessageHandler(
		Prio:=2, 								(*1=highest, .. , 4=lowest*)
		Btn1Addr:=ADR(MsgOk),				(*Address of Button1 , if Zero then Button is unvisible*)
		Btn2Addr:=ADR(MsgCancel),			(*Address of Button2 , if Zero then Button is unvisible*)
		sVisu:=Visu.Message);
END_ACTION

ACTION Msg_Cam2_exit:
MsgOk:=FALSE;
MsgCancel:=FALSE;
END_ACTION

ACTION Cam2_CounterReset_entry:
NokCounter_Cam[2] := 0;
NokCounterPercent_Cam[2] := 0;
(*Percent Register löschen*)
FOR i:=1 TO 100 BY 1 DO
  NokPercent_Cam[2,i]:= FALSE;
END_FOR
END_ACTION

ACTION Cam2_WaitRepeat_entry:
Delay(IN:=FALSE);
END_ACTION

ACTION Cam2_WaitRepeat_action:
Delay(	IN:=TRUE, 		(*warte kurz, bevor neues Bild gemacht wird *)
		PT:=T#750ms);
END_ACTION

ACTION Cam2_ResultOK_entry:
Result_Cam2 := RESULT_OK;
END_ACTION

ACTION Result_Total_entry:
IF	Result_Cam1[1] = RESULT_OK AND
	Result_Cam1[2] = RESULT_OK AND
	Result_Cam2 = RESULT_OK THEN
	Result := RESULT_OK;
ELSE
	Result := RESULT_NOK;
	gNokPartsColorCam := gNokPartsColorCam + 1;
END_IF
END_ACTION

ACTION ResetLock_entry:
LockForCam:=FALSE;
END_ACTION

ACTION SeqEnd_action:
SFCTime:=TIME_TO_DINT(TIME()-SFCTimeStart);
State:=STATE_WAIT;
END_ACTION

TRANSITION Kamera_betriebsbereit:
(*Kamera betriebsbereit oder nicht Aktiv*)

(* Sensopart Kamera *)
(NOT ST03_8_100_A1.Activated OR
ST03_8_100_A1.Activated AND
NOT ST03_8_100_A1.sm_kamera_nicht_bb) AND
(* Keyence Kamera *)
(NOT ST03_8_105_A1.sConfig.Aktiv OR
ST03_8_105_A1.sConfig.Aktiv AND
NOT ST03_8_105_A1.sm_kamera_nicht_bb)
END_TRANSITION

TRANSITION Done:
Delay.Q
END_TRANSITION

TRANSITION Check_Part:
Robot01.ActualArea <> 4 AND (
NOT ST03_4x3_B70_0.BitInToCheck OR	(* ISK anwesend Übergabeposition Stopper*)
NOT ST03_4x3_B70_1.BitInToCheck )	(* ISK anwesend Übergabeposition*)
END_TRANSITION

TRANSITION PosEmpty:
NOT ST03_4x2_B69_5.BitInToCheck			 	(*  ISK anwesend am Stopper*)
END_TRANSITION

TRANSITION State Ok:
ST03_4x3_Y70_5.State=STATE_OK (*Zuführung Vereinzler AST/GST *)
END_TRANSITION

TRANSITION Part Ready:
Delay.Q
END_TRANSITION

TRANSITION PosFull:
ST03_4x2_B69_5.BitInToCheck			 	(*  ISK anwesend am Stopper*)
END_TRANSITION

TRANSITION State Ok:
ST03_4x3_Y70_5.State=STATE_OK (*Zuführung Vereinzler AST/GST *)
END_TRANSITION

TRANSITION Pos1Empty:
NOT ST03_4x3_B70_0.BitInToCheck AND 	(*  ISK anwesend Übergabeposition Stopper*)
ST03_4x2_B69_5.BitInToCheck			 	(*  ISK anwesend am Stopper*)
END_TRANSITION

TRANSITION State Ok:
ST03_4x3_Y70_6.State=STATE_OK 	(*Zuführung Stopper AST/GST *)
END_TRANSITION

TRANSITION Pos2Empty:
ST03_4x3_B70_0.BitInToCheck AND 	(*  ISK anwesend Übergabeposition Stopper*)
NOT ST03_4x3_B70_1.BitInToCheck AND 	(*  ISK anwesend Übergabeposition*)
ST03_4x2_B69_5.BitInToCheck			 	(*  ISK anwesend am Stopper*)
END_TRANSITION

TRANSITION Part Ready:
Delay.Q
END_TRANSITION

TRANSITION Pos1Full:
ST03_4x3_B70_0.BitInToCheck 	(*ISK anwesend Übergabeposition Stopper*)
END_TRANSITION

TRANSITION State Ok:
ST03_4x3_Y70_6.State=STATE_OK AND	(*Zuführung Stopper AST/GST *)
ST03_4x3_Y70_5.State=STATE_OK (*Zuführung Vereinzler AST/GST *)
END_TRANSITION

TRANSITION Cam1Active:
ST03_8_105_A1.sConfig.Aktiv
END_TRANSITION

TRANSITION Busy:
ST03_8_105_A1.st_ctrl_out.b_busy	 (*Kamera Ehternet*)
END_TRANSITION

TRANSITION Done:
ST03_8_105_A1.st_ctrl_out.b_fertig
END_TRANSITION

TRANSITION result_ok:
Result_Cam1[Part] = RESULT_OK OR
RepeatCounter >= 2
END_TRANSITION

TRANSITION Repeat_:
TRUE
END_TRANSITION

TRANSITION Done:
Delay.Q
END_TRANSITION

TRANSITION Cam1_CounterOK:
NokCounter_Cam[1] < MP.ST03.CamNoOfErrors_KYE AND
NokCounterPercent_Cam[1] < MP.ST03.CamNoOfErrorsPercent_KYE
END_TRANSITION

TRANSITION Cam1_Nok:
NokCounter_Cam[1] >= MP.ST03.CamNoOfErrors_KYE OR
NokCounterPercent_Cam[1] >= MP.ST03.CamNoOfErrorsPercent_KYE
END_TRANSITION

TRANSITION NotActive:
TRUE
END_TRANSITION

TRANSITION Tippbetrieb:
gTipImp
END_TRANSITION

TRANSITION Pos2Empty:
NOT ST03_4x3_B70_1.BitInToCheck AND 	(*  ISK anwesend Übergabeposition*)
ST03_4x3_B70_0.BitInToCheck			 	(*  ISK anwesend Übergabeposition Stopper*)
END_TRANSITION

TRANSITION State Ok:
ST03_4x3_Y70_7.State=STATE_OK 	(* Zuführung Stopper Übergabeposition AST/GST *)
END_TRANSITION

TRANSITION Part Ready:
Delay.Q
END_TRANSITION

TRANSITION Pos2Full:
ST03_4x3_B70_1.BitInToCheck	 	(*ISK anwesend Übergabeposition*)
END_TRANSITION

TRANSITION State Ok:
ST03_4x3_Y70_7.State=STATE_OK 	(* Zuführung Stopper Übergabeposition AST/GST *)
END_TRANSITION

TRANSITION Pos12Full:
ST03_4x3_B70_0.BitInToCheck AND		(*  ISK anwesend Übergabeposition 1*)
ST03_4x3_B70_1.BitInToCheck		 	(*  ISK anwesend Übergabeposition 2*)
END_TRANSITION

TRANSITION Cam2Active:
ST03_8_100_A1.Activated
END_TRANSITION

TRANSITION Busy:
ST03_8_100_A1.st_ctrl_out.b_busy 	(*Kamera Farberkennung Ehternet*)
END_TRANSITION

TRANSITION Done:
ST03_8_100_A1.st_ctrl_out.b_fertig
END_TRANSITION

TRANSITION result_ok:
Result_Cam2 = RESULT_OK OR
RepeatCounter >= 2
END_TRANSITION

TRANSITION Cam2_CounterOK:
NokCounter_Cam[2] < MP.ST03.CamNoOfErrors AND
NokCounterPercent_Cam[2] < MP.ST03.CamNoOfErrorsPercent
END_TRANSITION

TRANSITION Cam2_Nok:
NokCounter_Cam[2] >= MP.ST03.CamNoOfErrors OR
NokCounterPercent_Cam[2] >= MP.ST03.CamNoOfErrorsPercent
END_TRANSITION

TRANSITION Repeat_:
TRUE
END_TRANSITION

TRANSITION Done:
Delay.Q
END_TRANSITION

TRANSITION NotActive:
TRUE
END_TRANSITION

TRANSITION Tippbetrieb:
gTipImp
END_TRANSITION
END_PROGRAM

(* POU Stations/ST_00/ST00_SFCs/_SpecialModeSFCs/CallSpecialModeSFCs, ST *)
PROGRAM CallSpecialModeSFCs
VAR_OUTPUT
  AllSpecialModeSFCInInit : BOOL := TRUE;

END_VAR
SpecialModeMain();
SpecialMode01();
SpecialMode02();
SpecialMode03();
SpecialMode04();
SpecialMode05();
SpecialMode06();
SpecialMode07();
SpecialMode08();

AllSpecialModeSFCInInit:=SpecialModeMain.State=STATE_OK;
END_PROGRAM

(* POU Stations/ST_00/ST00_SFCs/_SpecialModeSFCs/SpecialModeMain, SFC *)
PROGRAM SpecialModeMain
(* 09.MAY 2005 Ext/g.baiz *)

VAR_OUTPUT
	SFCCurrentPOU		: STRING:='SpecialModeMain';
	SFCCurrentStep	: STRING:='';
	SFCTime					:	DINT;
  State   				:	DINT;
  Result  				:	DINT;
END_VAR
VAR_INPUT
	ModeNo					: DINT;
END_VAR
VAR
	MsgOK				:	BOOL;
	MsgCancel		:	BOOL;
	SFCRun					:	BOOL;
	SFCTimeStart		:	TIME;
	(* Userdefinded area *)
	SpecMode01Flag	:	R_TRIG;
	SpecMode02Flag	:	R_TRIG;
	SpecMode03Flag	:	R_TRIG;
	SpecMode04Flag	:	R_TRIG;
	SpecMode05Flag	:	R_TRIG;
	SpecMode06Flag	:	R_TRIG;
	SpecMode07Flag	:	R_TRIG;
	SpecMode08Flag	:	R_TRIG;

	idx							:	INT;

END_VAR
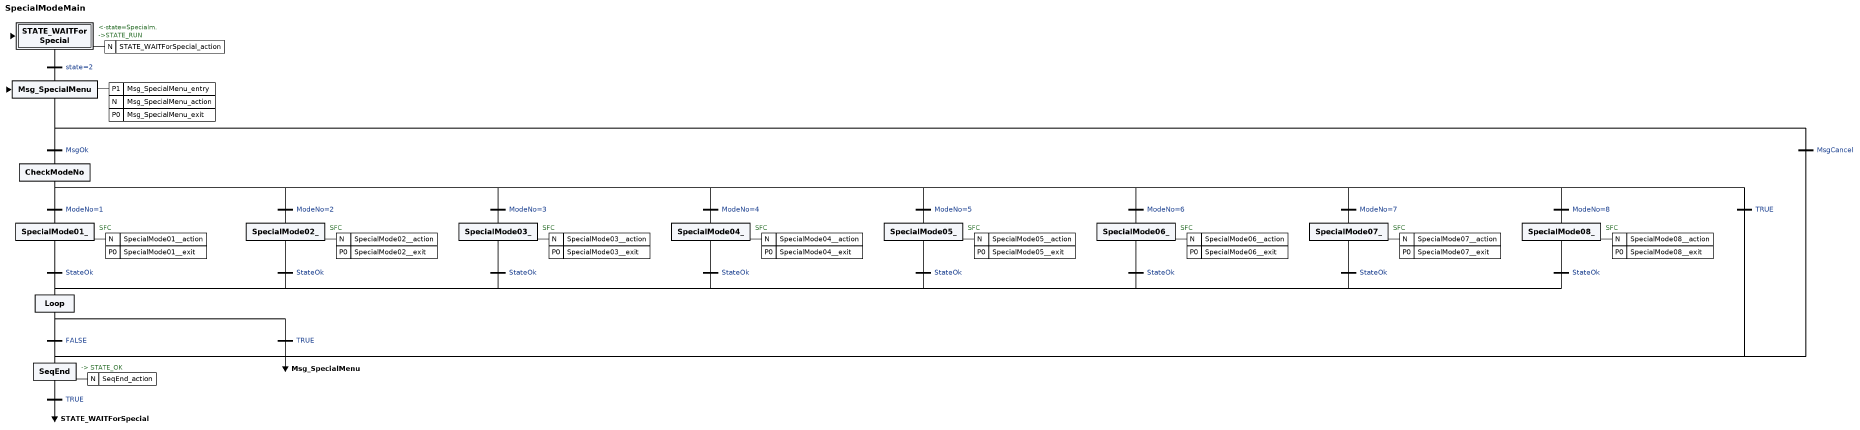
INITIAL_STEP STATE_WAITForSpecial: (* <-state=Specialm. / ->STATE_RUN *)
	STATE_WAITForSpecial_action(N);
END_STEP
TRANSITION FROM STATE_WAITForSpecial TO Msg_SpecialMenu := state=2;
END_TRANSITION
STEP Msg_SpecialMenu:
	Msg_SpecialMenu_entry(P1);
	Msg_SpecialMenu_action(N);
	Msg_SpecialMenu_exit(P0);
END_STEP
TRANSITION FROM Msg_SpecialMenu TO CheckModeNo := MsgOk;
END_TRANSITION
TRANSITION FROM Msg_SpecialMenu TO SeqEnd := MsgCancel;
END_TRANSITION
STEP CheckModeNo:
END_STEP
TRANSITION FROM CheckModeNo TO SpecialMode01_ := ModeNo=1;
END_TRANSITION
TRANSITION FROM CheckModeNo TO SpecialMode02_ := ModeNo=2;
END_TRANSITION
TRANSITION FROM CheckModeNo TO SpecialMode03_ := ModeNo=3;
END_TRANSITION
TRANSITION FROM CheckModeNo TO SpecialMode04_ := ModeNo=4;
END_TRANSITION
TRANSITION FROM CheckModeNo TO SpecialMode05_ := ModeNo=5;
END_TRANSITION
TRANSITION FROM CheckModeNo TO SpecialMode06_ := ModeNo=6;
END_TRANSITION
TRANSITION FROM CheckModeNo TO SpecialMode07_ := ModeNo=7;
END_TRANSITION
TRANSITION FROM CheckModeNo TO SpecialMode08_ := ModeNo=8;
END_TRANSITION
TRANSITION FROM CheckModeNo TO SeqEnd := TRUE;
END_TRANSITION
STEP SpecialMode01_: (* SFC *)
	SpecialMode01__action(N);
	SpecialMode01__exit(P0);
END_STEP
TRANSITION FROM SpecialMode01_ TO Loop := StateOk;
END_TRANSITION
STEP SpecialMode02_: (* SFC *)
	SpecialMode02__action(N);
	SpecialMode02__exit(P0);
END_STEP
TRANSITION FROM SpecialMode02_ TO Loop := StateOk;
END_TRANSITION
STEP SpecialMode03_: (* SFC *)
	SpecialMode03__action(N);
	SpecialMode03__exit(P0);
END_STEP
TRANSITION FROM SpecialMode03_ TO Loop := StateOk;
END_TRANSITION
STEP SpecialMode04_: (* SFC *)
	SpecialMode04__action(N);
	SpecialMode04__exit(P0);
END_STEP
TRANSITION FROM SpecialMode04_ TO Loop := StateOk;
END_TRANSITION
STEP SpecialMode05_: (* SFC *)
	SpecialMode05__action(N);
	SpecialMode05__exit(P0);
END_STEP
TRANSITION FROM SpecialMode05_ TO Loop := StateOk;
END_TRANSITION
STEP SpecialMode06_: (* SFC *)
	SpecialMode06__action(N);
	SpecialMode06__exit(P0);
END_STEP
TRANSITION FROM SpecialMode06_ TO Loop := StateOk;
END_TRANSITION
STEP SpecialMode07_: (* SFC *)
	SpecialMode07__action(N);
	SpecialMode07__exit(P0);
END_STEP
TRANSITION FROM SpecialMode07_ TO Loop := StateOk;
END_TRANSITION
STEP SpecialMode08_: (* SFC *)
	SpecialMode08__action(N);
	SpecialMode08__exit(P0);
END_STEP
TRANSITION FROM SpecialMode08_ TO Loop := StateOk;
END_TRANSITION
STEP Loop:
END_STEP
TRANSITION FROM Loop TO SeqEnd := FALSE;
END_TRANSITION
TRANSITION FROM Loop TO Msg_SpecialMenu := TRUE;
END_TRANSITION
STEP SeqEnd: (* -> STATE_OK *)
	SeqEnd_action(N);
END_STEP
TRANSITION FROM SeqEnd TO STATE_WAITForSpecial := TRUE;
END_TRANSITION

ACTION STATE_WAITForSpecial_action:
IF 	ModeSelect.Mode=MODE_SPECIAL
THEN
	State:=STATE_RUN;
	Result:=RESULT_NON;
	SFCTimeStart:=TIME();
ELSE
	State:=STATE_WAIT;
	SFCRun:=FALSE;
END_IF
END_ACTION

ACTION Msg_SpecialMenu_entry:
MessageHandler.ClearMessageLines(sVisu:=Visu.Message);

